C07300=1209.413,-55.510,-39.926,179.767,5.473,149.028
C07301=1209.418,-55.759,-39.914,179.765,5.472,149.029
C07302=1209.423,-56.009,-39.902,179.762,5.472,149.030
C07303=1209.429,-56.259,-39.890,179.760,5.472,149.030
C07304=1209.434,-56.509,-39.878,179.758,5.472,149.031
C07305=1209.439,-56.758,-39.867,179.755,5.471,149.032
C07306=1209.444,-57.008,-39.855,179.753,5.472,149.032
C07307=1209.449,-57.258,-39.843,179.750,5.471,149.033
C07308=1209.454,-57.508,-39.832,179.747,5.471,149.034
C07309=1209.459,-57.757,-39.819,179.745,5.471,149.035
C07310=1209.464,-58.007,-39.808,179.743,5.470,149.035
C07311=1209.470,-58.256,-39.796,179.741,5.471,149.036
C07312=1209.475,-58.506,-39.784,179.738,5.470,149.036
C07313=1209.480,-58.755,-39.773,179.736,5.470,149.037
C07314=1209.486,-59.005,-39.761,179.734,5.470,149.038
C07315=1209.491,-59.255,-39.748,179.731,5.470,149.039
C07316=1209.495,-59.504,-39.737,179.728,5.469,149.039
C07317=1209.501,-59.754,-39.725,179.726,5.470,149.040
C07318=1209.506,-60.004,-39.713,179.724,5.469,149.040
C07319=1209.511,-60.254,-39.702,179.722,5.469,149.041
C07320=1209.516,-60.504,-39.690,179.719,5.469,149.042
C07321=1209.522,-60.753,-39.679,179.717,5.468,149.043
C07322=1209.527,-61.003,-39.667,179.715,5.469,149.043
C07323=1209.533,-61.252,-39.656,179.712,5.468,149.044
C07324=1209.537,-61.501,-39.644,179.710,5.469,149.045
C07325=1209.542,-61.751,-39.632,179.707,5.468,149.045
C07326=1209.547,-62.001,-39.620,179.705,5.467,149.046
C07327=1209.552,-62.251,-39.608,179.703,5.468,149.047
C07328=1209.557,-62.501,-39.597,179.700,5.467,149.047
C07329=1209.563,-62.750,-39.586,179.698,5.468,149.048
C07330=1209.569,-63.000,-39.574,179.695,5.467,149.049
C07331=1209.573,-63.249,-39.562,179.693,5.467,149.049
C07332=1209.579,-63.499,-39.551,179.691,5.467,149.050
C07333=1209.583,-63.749,-39.539,179.688,5.467,149.051
C07334=1209.589,-63.999,-39.527,179.686,5.466,149.051
C07335=1209.594,-64.249,-39.516,179.684,5.466,149.052
C07336=1209.600,-64.498,-39.505,179.681,5.466,149.053
C07337=1209.604,-64.747,-39.493,179.679,5.466,149.053
C07338=1209.610,-64.997,-39.481,179.676,5.466,149.054
C07339=1209.614,-65.247,-39.470,179.674,5.466,149.055
C07340=1209.620,-65.497,-39.458,179.672,5.465,149.056
C07341=1209.625,-65.746,-39.447,179.669,5.465,149.056
C07342=1209.631,-65.996,-39.435,179.667,5.465,149.057
C07343=1209.635,-66.245,-39.424,179.665,5.464,149.057
C07344=1209.641,-66.495,-39.412,179.663,5.465,149.058
C07345=1209.646,-66.746,-39.402,179.660,5.464,149.059
C07346=1209.651,-66.996,-39.390,179.657,5.464,149.060
C07347=1209.656,-67.244,-39.379,179.655,5.464,149.060
C07348=1209.662,-67.494,-39.367,179.652,5.464,149.061
C07349=1209.667,-67.744,-39.356,179.650,5.464,149.062
C07350=1209.672,-67.994,-39.344,179.648,5.463,149.062
C07351=1209.677,-68.243,-39.333,179.646,5.463,149.063
C07352=1209.682,-68.492,-39.322,179.643,5.463,149.064
C07353=1209.687,-68.742,-39.310,179.641,5.463,149.064
C07354=1209.692,-68.993,-39.299,179.639,5.463,149.065
C07355=1209.698,-69.243,-39.287,179.636,5.463,149.066
C07356=1209.703,-69.492,-39.276,179.633,5.462,149.066
C07357=1209.709,-69.741,-39.264,179.632,5.462,149.067
C07358=1209.713,-69.991,-39.253,179.629,5.462,149.068
C07359=1209.718,-70.241,-39.242,179.627,5.462,149.068
C07360=1209.724,-70.491,-39.231,179.624,5.462,149.069
C07361=1209.729,-70.740,-39.220,179.622,5.462,149.070
C07362=1209.734,-70.990,-39.208,179.620,5.462,149.070
C07363=1209.739,-71.240,-39.197,179.617,5.461,149.071
C07364=1209.744,-71.489,-39.186,179.615,5.462,149.072
C07365=1209.750,-71.739,-39.175,179.613,5.461,149.072
C07366=1209.755,-71.989,-39.163,179.611,5.461,149.073
C07367=1209.761,-72.238,-39.152,179.608,5.461,149.074
C07368=1209.765,-72.488,-39.140,179.606,5.461,149.074
C07369=1209.770,-72.737,-39.129,179.603,5.461,149.075
C07370=1209.776,-72.988,-39.118,179.600,5.460,149.076
C07371=1209.781,-73.237,-39.107,179.598,5.461,149.077
C07372=1209.786,-73.486,-39.096,179.596,5.460,149.077
C07373=1209.792,-73.737,-39.085,179.594,5.460,149.078
C07374=1209.797,-73.986,-39.074,179.591,5.460,149.078
C07375=1209.802,-74.236,-39.062,179.589,5.460,149.079
C07376=1209.807,-74.485,-39.050,179.587,5.460,149.080
C07377=1209.813,-74.756,-39.039,179.584,5.459,149.081
C07378=1209.818,-75.026,-39.027,179.582,5.459,149.081
C07379=1209.824,-75.297,-39.015,179.579,5.459,149.082
C07380=1209.830,-75.568,-39.003,179.577,5.459,149.083
C07381=1209.835,-75.817,-38.992,179.575,5.459,149.083
C07382=1209.840,-76.068,-38.980,179.572,5.459,149.084
C07383=1209.846,-76.317,-38.969,179.569,5.458,149.085
C07384=1209.850,-76.566,-38.958,179.567,5.458,149.086
C07385=1209.855,-76.817,-38.948,179.565,5.458,149.086
C07386=1209.861,-77.066,-38.936,179.563,5.458,149.087
C07387=1209.866,-77.316,-38.925,179.560,5.458,149.087
C07388=1209.871,-77.566,-38.914,179.558,5.458,149.088
C07389=1209.877,-77.815,-38.903,179.555,5.457,149.089
C07390=1209.882,-78.065,-38.892,179.553,5.457,149.090
C07391=1209.887,-78.315,-38.881,179.551,5.457,149.090
C07392=1209.892,-78.564,-38.870,179.548,5.457,149.091
C07393=1209.897,-78.814,-38.859,179.546,5.457,149.091
C07394=1209.903,-79.064,-38.847,179.544,5.457,149.092
C07395=1209.908,-79.314,-38.837,179.542,5.457,149.093
C07396=1209.913,-79.563,-38.826,179.539,5.456,149.094
C07397=1209.918,-79.813,-38.816,179.537,5.457,149.094
C07398=1209.924,-80.063,-38.804,179.535,5.456,149.095
C07399=1209.929,-80.313,-38.793,179.532,5.456,149.095
C07400=1209.934,-80.562,-38.782,179.530,5.456,149.096
C07401=1209.939,-80.811,-38.771,179.527,5.455,149.097
C07402=1209.944,-81.061,-38.761,179.525,5.456,149.098
C07403=1209.950,-81.311,-38.749,179.522,5.455,149.098
C07404=1209.955,-81.561,-38.738,179.521,5.455,149.099
C07405=1209.960,-81.810,-38.727,179.518,5.455,149.099
C07406=1209.965,-82.060,-38.717,179.516,5.455,149.100
C07407=1209.970,-82.309,-38.706,179.513,5.455,149.101
C07408=1209.975,-82.559,-38.695,179.511,5.455,149.102
C07409=1209.981,-82.809,-38.683,179.509,5.455,149.102
C07410=1209.986,-83.059,-38.673,179.506,5.454,149.103
C07411=1209.991,-83.309,-38.663,179.504,5.454,149.104
C07412=1209.997,-83.558,-38.652,179.502,5.454,149.104
C07413=1210.002,-83.808,-38.641,179.500,5.454,149.105
C07414=1210.006,-84.058,-38.630,179.497,5.454,149.106
C07415=1210.012,-84.308,-38.620,179.495,5.454,149.106
C07416=1210.017,-84.557,-38.608,179.492,5.454,149.107
C07417=1210.023,-84.807,-38.598,179.491,5.454,149.108
C07418=1210.028,-85.057,-38.587,179.488,5.453,149.108
C07419=1210.033,-85.306,-38.576,179.486,5.454,149.109
C07420=1210.038,-85.556,-38.566,179.483,5.453,149.110
C07421=1210.044,-85.805,-38.555,179.481,5.453,149.110
C07422=1210.049,-86.056,-38.544,179.478,5.453,149.111
C07423=1210.054,-86.306,-38.533,179.476,5.452,149.112
C07424=1210.059,-86.555,-38.523,179.474,5.453,149.112
C07425=1210.064,-86.805,-38.512,179.471,5.452,149.113
C07426=1210.069,-87.054,-38.501,179.469,5.453,149.114
C07427=1210.074,-87.304,-38.490,179.467,5.452,149.114
C07428=1210.080,-87.554,-38.480,179.465,5.452,149.115
C07429=1210.085,-87.804,-38.468,179.462,5.452,149.116
C07430=1210.091,-88.053,-38.458,179.460,5.452,149.116
C07431=1210.096,-88.303,-38.448,179.458,5.452,149.117
C07432=1210.101,-88.552,-38.437,179.456,5.452,149.118
C07433=1210.106,-88.803,-38.426,179.453,5.452,149.118
C07434=1210.112,-89.052,-38.416,179.451,5.451,149.119
C07435=1210.117,-89.302,-38.405,179.449,5.451,149.120
C07436=1210.122,-89.551,-38.394,179.446,5.451,149.120
C07437=1210.127,-89.802,-38.384,179.444,5.451,149.121
C07438=1210.133,-90.051,-38.374,179.441,5.451,149.122
C07439=1210.137,-90.301,-38.362,179.439,5.451,149.122
C07440=1210.143,-90.550,-38.352,179.437,5.450,149.123
C07441=1210.148,-90.801,-38.341,179.435,5.451,149.124
C07442=1210.154,-91.050,-38.331,179.432,5.450,149.124
C07443=1210.158,-91.300,-38.320,179.430,5.451,149.125
C07444=1210.164,-91.549,-38.310,179.427,5.450,149.126
C07445=1210.169,-91.800,-38.299,179.426,5.450,149.126
C07446=1210.174,-92.049,-38.289,179.423,5.450,149.127
C07447=1210.179,-92.299,-38.278,179.421,5.450,149.128
C07448=1210.185,-92.548,-38.268,179.418,5.450,149.128
C07449=1210.190,-92.798,-38.257,179.416,5.450,149.129
C07450=1210.195,-93.048,-38.247,179.414,5.449,149.130
C07451=1210.200,-93.297,-38.237,179.412,5.450,149.130
C07452=1210.205,-93.547,-38.227,179.409,5.449,149.131
C07453=1210.210,-93.796,-38.216,179.407,5.449,149.132
C07454=1210.215,-94.047,-38.205,179.405,5.449,149.132
C07455=1210.221,-94.296,-38.195,179.402,5.449,149.133
C07456=1210.226,-94.546,-38.184,179.400,5.449,149.134
C07457=1210.232,-94.796,-38.174,179.398,5.448,149.134
C07458=1210.237,-95.046,-38.164,179.396,5.449,149.135
C07459=1210.242,-95.296,-38.153,179.393,5.448,149.136
C07460=1210.248,-95.545,-38.142,179.391,5.449,149.137
C07461=1210.253,-95.795,-38.132,179.389,5.448,149.137
C07462=1210.258,-96.044,-38.122,179.387,5.448,149.138
C07463=1210.263,-96.294,-38.112,179.384,5.448,149.138
C07464=1210.268,-96.544,-38.101,179.382,5.448,149.139
C07465=1210.274,-96.793,-38.091,179.379,5.448,149.140
C07466=1210.279,-97.044,-38.081,179.377,5.448,149.140
C07467=1210.284,-97.293,-38.070,179.375,5.447,149.141
C07468=1210.290,-97.543,-38.060,179.373,5.448,149.142
C07469=1210.295,-97.793,-38.050,179.370,5.447,149.142
C07470=1210.300,-98.043,-38.039,179.368,5.448,149.143
C07471=1210.305,-98.293,-38.029,179.366,5.447,149.144
C07472=1210.310,-98.541,-38.018,179.364,5.447,149.144
C07473=1210.316,-98.791,-38.008,179.361,5.447,149.145
C07474=1210.321,-99.041,-37.998,179.359,5.447,149.146
C07475=1210.326,-99.291,-37.987,179.357,5.446,149.146
C07476=1210.332,-99.540,-37.977,179.355,5.447,149.147
C07477=1210.336,-99.790,-37.967,179.352,5.446,149.148
C07478=1210.342,-100.040,-37.957,179.350,5.447,149.148
C07479=1210.347,-100.289,-37.947,179.347,5.446,149.149
C07480=1210.352,-100.540,-37.936,179.346,5.446,149.150
C07481=1210.357,-100.811,-37.925,179.343,5.446,149.150
C07482=1210.364,-101.082,-37.914,179.340,5.445,149.151
C07483=1210.369,-101.353,-37.903,179.338,5.446,149.152
C07484=1210.375,-101.625,-37.892,179.335,5.446,149.153
C07485=1210.380,-101.875,-37.883,179.333,5.446,149.153
C07486=1210.386,-102.124,-37.873,179.331,5.445,149.154
C07487=1210.391,-102.374,-37.862,179.329,5.446,149.155
C07488=1210.396,-102.624,-37.852,179.326,5.445,149.155
C07489=1210.401,-102.873,-37.842,179.324,5.445,149.156
C07490=1210.406,-103.123,-37.832,179.322,5.445,149.157
C07491=1210.412,-103.373,-37.821,179.320,5.445,149.157
C07492=1210.417,-103.622,-37.811,179.317,5.445,149.158
C07493=1210.422,-103.872,-37.801,179.315,5.445,149.159
C07494=1210.427,-104.122,-37.791,179.313,5.444,149.159
C07495=1210.433,-104.371,-37.781,179.311,5.445,149.160
C07496=1210.438,-104.622,-37.771,179.308,5.444,149.161
C07497=1210.443,-104.872,-37.761,179.306,5.445,149.161
C07498=1210.449,-105.121,-37.751,179.304,5.444,149.162
C07499=1210.454,-105.371,-37.741,179.302,5.444,149.162
C07500=1210.458,-105.621,-37.731,179.299,5.444,149.163
C07501=1210.464,-105.870,-37.721,179.297,5.444,149.164
C07502=1210.470,-106.120,-37.711,179.295,5.444,149.164
C07503=1210.475,-106.371,-37.701,179.292,5.444,149.165
C07504=1210.480,-106.620,-37.691,179.290,5.444,149.166
C07505=1210.485,-106.869,-37.681,179.288,5.444,149.167
C07506=1210.491,-107.119,-37.671,179.285,5.444,149.167
C07507=1210.495,-107.369,-37.661,179.283,5.444,149.168
C07508=1210.501,-107.618,-37.650,179.281,5.443,149.168
C07509=1210.507,-107.869,-37.641,179.279,5.443,149.169
C07510=1210.512,-108.118,-37.631,179.276,5.443,149.170
C07511=1210.517,-108.368,-37.621,179.274,5.443,149.170
C07512=1210.522,-108.618,-37.611,179.272,5.443,149.171
C07513=1210.527,-108.867,-37.602,179.270,5.443,149.172
C07514=1210.533,-109.117,-37.591,179.267,5.443,149.173
C07515=1210.537,-109.367,-37.581,179.265,5.443,149.173
C07516=1210.543,-109.616,-37.571,179.263,5.442,149.174
C07517=1210.549,-109.867,-37.562,179.261,5.443,149.174
C07518=1210.554,-110.116,-37.552,179.258,5.442,149.175
C07519=1210.559,-110.365,-37.542,179.256,5.442,149.176
C07520=1210.564,-110.616,-37.531,179.254,5.442,149.176
C07521=1210.569,-110.865,-37.522,179.252,5.442,149.177
C07522=1210.575,-111.115,-37.512,179.249,5.442,149.178
C07523=1210.580,-111.364,-37.503,179.247,5.442,149.178
C07524=1210.585,-111.615,-37.493,179.245,5.441,149.179
C07525=1210.591,-111.865,-37.483,179.242,5.442,149.180
C07526=1210.596,-112.114,-37.473,179.240,5.441,149.180
C07527=1210.602,-112.364,-37.463,179.238,5.441,149.181
C07528=1210.606,-112.613,-37.454,179.236,5.441,149.182
C07529=1210.612,-112.863,-37.444,179.233,5.441,149.182
C07530=1210.617,-113.113,-37.434,179.231,5.441,149.183
C07531=1210.622,-113.363,-37.424,179.229,5.441,149.184
C07532=1210.628,-113.612,-37.414,179.227,5.441,149.184
C07533=1210.633,-113.862,-37.405,179.224,5.441,149.185
C07534=1210.639,-114.112,-37.395,179.222,5.441,149.186
C07535=1210.643,-114.362,-37.385,179.220,5.440,149.186
C07536=1210.649,-114.612,-37.375,179.218,5.441,149.187
C07537=1210.654,-114.861,-37.366,179.215,5.440,149.188
C07538=1210.659,-115.111,-37.356,179.213,5.441,149.188
C07539=1210.664,-115.361,-37.347,179.211,5.440,149.189
C07540=1210.670,-115.610,-37.336,179.209,5.440,149.189
C07541=1210.675,-115.860,-37.328,179.206,5.440,149.190
C07542=1210.680,-116.110,-37.317,179.205,5.440,149.191
C07543=1210.685,-116.360,-37.308,179.202,5.440,149.191
C07544=1210.691,-116.610,-37.298,179.200,5.440,149.192
C07545=1210.696,-116.859,-37.289,179.197,5.440,149.193
C07546=1210.702,-117.109,-37.279,179.196,5.440,149.193
C07547=1210.707,-117.359,-37.270,179.193,5.439,149.194
C07548=1210.712,-117.608,-37.260,179.191,5.440,149.195
C07549=1210.717,-117.858,-37.250,179.188,5.439,149.195
C07550=1210.723,-118.108,-37.240,179.187,5.439,149.196
C07551=1210.727,-118.358,-37.231,179.184,5.440,149.197
C07552=1210.733,-118.608,-37.221,179.182,5.439,149.197
C07553=1210.738,-118.857,-37.212,179.180,5.439,149.198
C07554=1210.743,-119.107,-37.203,179.178,5.439,149.199
C07555=1210.749,-119.356,-37.192,179.175,5.439,149.199
C07556=1210.754,-119.606,-37.183,179.173,5.439,149.200
C07557=1210.760,-119.856,-37.173,179.171,5.439,149.201
C07558=1210.764,-120.106,-37.164,179.168,5.438,149.201
C07559=1210.770,-120.357,-37.155,179.166,5.439,149.202
C07560=1210.775,-120.606,-37.145,179.164,5.438,149.202
C07561=1210.780,-120.856,-37.136,179.162,5.438,149.203
C07562=1210.786,-121.105,-37.126,179.159,5.438,149.204
C07563=1210.791,-121.355,-37.117,179.157,5.438,149.205
C07564=1210.797,-121.605,-37.107,179.155,5.437,149.205
C07565=1210.802,-121.854,-37.098,179.153,5.438,149.206
C07566=1210.807,-122.104,-37.088,179.151,5.438,149.207
C07567=1210.812,-122.354,-37.079,179.149,5.437,149.207
C07568=1210.818,-122.604,-37.070,179.147,5.438,149.208
C07569=1210.823,-122.853,-37.060,179.144,5.437,149.208
C07570=1210.828,-123.103,-37.051,179.142,5.437,149.209
C07571=1210.833,-123.354,-37.041,179.140,5.437,149.210
C07572=1210.839,-123.603,-37.031,179.138,5.437,149.210
C07573=1210.844,-123.853,-37.022,179.135,5.437,149.211
C07574=1210.849,-124.102,-37.013,179.133,5.437,149.212
C07575=1210.854,-124.352,-37.003,179.131,5.437,149.212
C07576=1210.860,-124.602,-36.994,179.129,5.437,149.213
C07577=1210.865,-124.852,-36.985,179.126,5.436,149.213
C07578=1210.870,-125.102,-36.975,179.124,5.437,149.214
C07579=1210.876,-125.352,-36.966,179.122,5.437,149.215
C07580=1210.880,-125.601,-36.957,179.120,5.436,149.215
C07581=1210.886,-125.851,-36.947,179.118,5.437,149.216
C07582=1210.892,-126.101,-36.938,179.115,5.436,149.217
C07583=1210.896,-126.350,-36.929,179.113,5.437,149.218
C07584=1210.902,-126.600,-36.919,179.111,5.436,149.218
C07585=1210.481,-126.611,-36.957,179.107,5.439,149.220
C07586=1210.476,-126.361,-36.966,179.109,5.440,149.219
C07587=1210.471,-126.111,-36.976,179.111,5.439,149.219
C07588=1210.465,-125.861,-36.985,179.113,5.440,149.218
C07589=1210.460,-125.611,-36.994,179.116,5.440,149.217
C07590=1210.455,-125.362,-37.004,179.118,5.440,149.217
C07591=1210.449,-125.112,-37.013,179.120,5.440,149.216
C07592=1210.444,-124.862,-37.022,179.122,5.440,149.216
C07593=1210.439,-124.613,-37.032,179.125,5.440,149.215
C07594=1210.433,-124.363,-37.041,179.127,5.440,149.214
C07595=1210.428,-124.113,-37.050,179.129,5.441,149.214
C07596=1210.423,-123.864,-37.060,179.131,5.440,149.213
C07597=1210.417,-123.614,-37.069,179.134,5.441,149.212
C07598=1210.412,-123.364,-37.078,179.135,5.441,149.212
C07599=1210.407,-123.114,-37.088,179.138,5.441,149.211
C07600=1210.401,-122.864,-37.097,179.140,5.441,149.210
C07601=1210.396,-122.614,-37.106,179.142,5.441,149.210
C07602=1210.390,-122.365,-37.116,179.144,5.441,149.209
C07603=1210.385,-122.115,-37.125,179.147,5.441,149.208
C07604=1210.380,-121.866,-37.135,179.149,5.441,149.208
C07605=1210.374,-121.616,-37.144,179.151,5.441,149.207
C07606=1210.369,-121.366,-37.154,179.153,5.441,149.206
C07607=1210.365,-121.116,-37.163,179.155,5.441,149.206
C07608=1210.359,-120.866,-37.173,179.158,5.442,149.205
C07609=1210.354,-120.616,-37.182,179.160,5.441,149.205
C07610=1210.348,-120.366,-37.192,179.162,5.442,149.204
C07611=1210.343,-120.117,-37.201,179.165,5.441,149.203
C07612=1210.337,-119.867,-37.211,179.167,5.442,149.203
C07613=1210.333,-119.618,-37.221,179.169,5.442,149.202
C07614=1210.327,-119.368,-37.229,179.172,5.442,149.201
C07615=1210.322,-119.118,-37.240,179.173,5.442,149.201
C07616=1210.317,-118.868,-37.249,179.176,5.443,149.200
C07617=1210.311,-118.619,-37.259,179.178,5.442,149.199
C07618=1210.307,-118.368,-37.268,179.181,5.443,149.199
C07619=1210.301,-118.119,-37.278,179.182,5.443,149.198
C07620=1210.296,-117.869,-37.287,179.184,5.442,149.197
C07621=1210.290,-117.619,-37.297,179.187,5.443,149.197
C07622=1210.285,-117.370,-37.306,179.189,5.443,149.196
C07623=1210.280,-117.120,-37.316,179.191,5.443,149.195
C07624=1210.274,-116.870,-37.325,179.193,5.443,149.195
C07625=1210.269,-116.621,-37.335,179.196,5.443,149.194
C07626=1210.264,-116.370,-37.345,179.198,5.443,149.194
C07627=1210.259,-116.121,-37.354,179.200,5.444,149.193
C07628=1210.254,-115.871,-37.365,179.202,5.443,149.192
C07629=1210.248,-115.621,-37.374,179.205,5.444,149.192
C07630=1210.243,-115.372,-37.384,179.207,5.444,149.191
C07631=1210.238,-115.122,-37.393,179.209,5.444,149.190
C07632=1210.233,-114.872,-37.403,179.211,5.444,149.189
C07633=1210.227,-114.622,-37.413,179.214,5.444,149.189
C07634=1210.222,-114.372,-37.422,179.216,5.444,149.188
C07635=1210.216,-114.123,-37.433,179.218,5.444,149.188
C07636=1210.211,-113.873,-37.441,179.220,5.444,149.187
C07637=1210.206,-113.623,-37.452,179.223,5.445,149.186
C07638=1210.201,-113.374,-37.461,179.225,5.444,149.186
C07639=1210.195,-113.123,-37.471,179.227,5.445,149.185
C07640=1210.191,-112.874,-37.481,179.229,5.444,149.184
C07641=1210.185,-112.624,-37.490,179.231,5.444,149.184
C07642=1210.179,-112.374,-37.500,179.234,5.445,149.183
C07643=1210.174,-112.125,-37.510,179.236,5.444,149.182
C07644=1210.169,-111.874,-37.520,179.239,5.445,149.182
C07645=1210.164,-111.625,-37.530,179.240,5.445,149.181
C07646=1210.158,-111.376,-37.540,179.243,5.445,149.180
C07647=1210.154,-111.126,-37.549,179.245,5.445,149.180
C07648=1210.148,-110.876,-37.559,179.247,5.446,149.179
C07649=1210.143,-110.626,-37.569,179.249,5.445,149.178
C07650=1210.138,-110.377,-37.579,179.252,5.446,149.178
C07651=1210.132,-110.127,-37.589,179.254,5.445,149.177
C07652=1210.127,-109.877,-37.598,179.256,5.446,149.177
C07653=1210.122,-109.627,-37.609,179.258,5.446,149.176
C07654=1210.116,-109.378,-37.619,179.261,5.446,149.175
C07655=1210.111,-109.128,-37.628,179.263,5.446,149.174
C07656=1210.106,-108.878,-37.638,179.265,5.447,149.174
C07657=1210.100,-108.629,-37.648,179.267,5.446,149.173
C07658=1210.096,-108.379,-37.658,179.270,5.447,149.172
C07659=1210.090,-108.128,-37.668,179.272,5.446,149.172
C07660=1210.084,-107.879,-37.678,179.275,5.447,149.171
C07661=1210.079,-107.630,-37.688,179.276,5.447,149.171
C07662=1210.074,-107.379,-37.698,179.279,5.447,149.170
C07663=1210.069,-107.130,-37.708,179.281,5.447,149.169
C07664=1210.064,-106.880,-37.717,179.284,5.447,149.168
C07665=1210.058,-106.631,-37.727,179.285,5.447,149.168
C07666=1210.053,-106.380,-37.738,179.288,5.448,149.167
C07667=1210.048,-106.131,-37.748,179.290,5.447,149.167
C07668=1210.043,-105.882,-37.758,179.293,5.448,149.166
C07669=1210.037,-105.631,-37.768,179.294,5.448,149.165
C07670=1210.032,-105.381,-37.777,179.297,5.448,149.165
C07671=1210.027,-105.132,-37.788,179.299,5.448,149.164
C07672=1210.021,-104.882,-37.798,179.302,5.448,149.163
C07673=1210.017,-104.632,-37.808,179.303,5.448,149.163
C07674=1210.011,-104.383,-37.818,179.306,5.448,149.162
C07675=1210.006,-104.133,-37.828,179.308,5.448,149.161
C07676=1210.001,-103.883,-37.839,179.311,5.448,149.161
C07677=1209.996,-103.633,-37.848,179.313,5.448,149.160
C07678=1209.990,-103.384,-37.858,179.315,5.449,149.159
C07679=1209.985,-103.133,-37.868,179.317,5.448,149.159
C07680=1209.979,-102.884,-37.879,179.320,5.449,149.158
C07681=1209.975,-102.635,-37.888,179.322,5.449,149.157
C07682=1209.970,-102.384,-37.899,179.324,5.449,149.157
C07683=1209.964,-102.135,-37.909,179.326,5.449,149.156
C07684=1209.958,-101.885,-37.919,179.329,5.449,149.155
C07685=1209.954,-101.635,-37.929,179.331,5.449,149.155
C07686=1209.948,-101.364,-37.940,179.334,5.449,149.154
C07687=1209.942,-101.093,-37.951,179.336,5.449,149.153
C07688=1209.936,-100.822,-37.963,179.338,5.449,149.152
C07689=1209.931,-100.551,-37.973,179.341,5.450,149.152
C07690=1209.926,-100.301,-37.984,179.343,5.449,149.151
C07691=1209.920,-100.051,-37.994,179.345,5.450,149.151
C07692=1209.915,-99.802,-38.004,179.348,5.450,149.150
C07693=1209.910,-99.552,-38.014,179.350,5.450,149.149
C07694=1209.905,-99.302,-38.025,179.352,5.450,149.148
C07695=1209.900,-99.052,-38.035,179.355,5.450,149.148
C07696=1209.894,-98.802,-38.045,179.357,5.450,149.147
C07697=1209.888,-98.553,-38.056,179.359,5.451,149.146
C07698=1209.884,-98.303,-38.066,179.361,5.450,149.146
C07699=1209.879,-98.053,-38.076,179.364,5.451,149.145
C07700=1209.873,-97.804,-38.086,179.366,5.451,149.145
C07701=1209.868,-97.554,-38.097,179.368,5.451,149.144
C07702=1209.862,-97.304,-38.107,179.370,5.451,149.143
C07703=1209.857,-97.054,-38.117,179.373,5.451,149.142
C07704=1209.852,-96.804,-38.128,179.375,5.451,149.142
C07705=1209.846,-96.555,-38.138,179.377,5.452,149.141
C07706=1209.842,-96.305,-38.148,179.379,5.451,149.141
C07707=1209.836,-96.055,-38.158,179.382,5.452,149.140
C07708=1209.831,-95.805,-38.168,179.384,5.451,149.139
C07709=1209.826,-95.556,-38.179,179.387,5.452,149.138
C07710=1209.820,-95.307,-38.190,179.388,5.452,149.138
C07711=1209.815,-95.056,-38.200,179.391,5.452,149.137
C07712=1209.810,-94.807,-38.210,179.393,5.452,149.136
C07713=1209.805,-94.556,-38.221,179.396,5.452,149.136
C07714=1209.799,-94.307,-38.231,179.399,5.453,149.135
C07715=1209.794,-94.057,-38.241,179.400,5.453,149.135
C07716=1209.789,-93.807,-38.252,179.403,5.453,149.134
C07717=1209.784,-93.559,-38.262,179.405,5.453,149.133
C07718=1209.779,-93.308,-38.273,179.408,5.453,149.132
C07719=1209.774,-93.059,-38.283,179.410,5.453,149.132
C07720=1209.769,-92.808,-38.294,179.412,5.454,149.131
C07721=1209.763,-92.559,-38.304,179.414,5.453,149.131
C07722=1209.758,-92.309,-38.315,179.417,5.454,149.130
C07723=1209.753,-92.060,-38.325,179.419,5.453,149.129
C07724=1209.747,-91.810,-38.336,179.421,5.454,149.128
C07725=1209.742,-91.560,-38.346,179.423,5.453,149.128
C07726=1209.736,-91.310,-38.356,179.426,5.454,149.127
C07727=1209.732,-91.061,-38.368,179.428,5.454,149.127
C07728=1209.726,-90.811,-38.378,179.430,5.454,149.126
C07729=1209.721,-90.561,-38.388,179.433,5.454,149.125
C07730=1209.716,-90.312,-38.399,179.435,5.454,149.124
C07731=1209.711,-90.062,-38.410,179.437,5.454,149.124
C07732=1209.705,-89.812,-38.420,179.439,5.455,149.123
C07733=1209.700,-89.562,-38.431,179.442,5.454,149.122
C07734=1209.695,-89.313,-38.441,179.444,5.455,149.122
C07735=1209.690,-89.063,-38.452,179.447,5.455,149.121
C07736=1209.684,-88.813,-38.462,179.448,5.455,149.121
C07737=1209.679,-88.563,-38.473,179.451,5.456,149.120
C07738=1209.674,-88.314,-38.484,179.453,5.455,149.119
C07739=1209.669,-88.064,-38.494,179.456,5.456,149.118
C07740=1209.663,-87.814,-38.505,179.458,5.455,149.118
C07741=1209.659,-87.565,-38.516,179.461,5.456,149.117
C07742=1209.653,-87.315,-38.526,179.462,5.456,149.117
C07743=1209.648,-87.065,-38.537,179.465,5.456,149.116
C07744=1209.643,-86.816,-38.548,179.467,5.456,149.115
C07745=1209.637,-86.566,-38.559,179.470,5.456,149.114
C07746=1209.632,-86.316,-38.569,179.472,5.456,149.114
C07747=1209.627,-86.066,-38.580,179.474,5.456,149.113
C07748=1209.622,-85.816,-38.591,179.477,5.457,149.112
C07749=1209.617,-85.567,-38.602,179.479,5.457,149.112
C07750=1209.612,-85.317,-38.612,179.481,5.457,149.111
C07751=1209.606,-85.067,-38.623,179.484,5.457,149.110
C07752=1209.601,-84.818,-38.634,179.486,5.457,149.110
C07753=1209.596,-84.568,-38.644,179.488,5.457,149.109
C07754=1209.591,-84.319,-38.655,179.490,5.458,149.108
C07755=1209.585,-84.069,-38.666,179.493,5.457,149.108
C07756=1209.580,-83.818,-38.677,179.495,5.458,149.107
C07757=1209.575,-83.569,-38.688,179.497,5.457,149.106
C07758=1209.569,-83.319,-38.698,179.500,5.458,149.106
C07759=1209.565,-83.070,-38.710,179.502,5.459,149.105
C07760=1209.559,-82.820,-38.720,179.504,5.458,149.104
C07761=1209.554,-82.571,-38.731,179.507,5.459,149.104
C07762=1209.549,-82.321,-38.741,179.509,5.458,149.103
C07763=1209.543,-82.071,-38.753,179.512,5.459,149.102
C07764=1209.538,-81.821,-38.764,179.514,5.458,149.102
C07765=1209.533,-81.572,-38.775,179.516,5.459,149.101
C07766=1209.528,-81.322,-38.785,179.518,5.459,149.100
C07767=1209.523,-81.073,-38.796,179.521,5.459,149.100
C07768=1209.518,-80.822,-38.807,179.523,5.460,149.099
C07769=1209.512,-80.573,-38.819,179.525,5.459,149.098
C07770=1209.507,-80.323,-38.829,179.528,5.460,149.098
C07771=1209.502,-80.073,-38.840,179.530,5.459,149.097
C07772=1209.497,-79.823,-38.851,179.532,5.460,149.096
C07773=1209.492,-79.574,-38.862,179.534,5.460,149.096
C07774=1209.486,-79.324,-38.873,179.537,5.460,149.095
C07775=1209.481,-79.075,-38.884,179.539,5.460,149.094
C07776=1209.476,-78.825,-38.895,179.542,5.460,149.094
C07777=1209.471,-78.575,-38.906,179.545,5.461,149.093
C07778=1209.465,-78.326,-38.917,179.546,5.461,149.092
C07779=1209.460,-78.075,-38.928,179.549,5.461,149.092
C07780=1209.455,-77.826,-38.939,179.551,5.461,149.091
C07781=1209.450,-77.577,-38.950,179.554,5.461,149.090
C07782=1209.444,-77.326,-38.961,179.556,5.461,149.090
C07783=1209.440,-77.077,-38.972,179.558,5.461,149.089
C07784=1209.434,-76.827,-38.983,179.560,5.462,149.088
C07785=1209.429,-76.577,-38.994,179.563,5.462,149.088
C07786=1209.424,-76.328,-39.006,179.565,5.462,149.087
C07787=1209.418,-76.078,-39.016,179.567,5.462,149.086
C07788=1209.414,-75.828,-39.027,179.570,5.462,149.085
C07789=1209.408,-75.579,-39.039,179.572,5.462,149.085
C07790=1209.403,-75.308,-39.050,179.575,5.463,149.084
C07791=1209.397,-75.037,-39.063,179.578,5.463,149.083
C07792=1209.391,-74.767,-39.075,179.580,5.463,149.083
C07793=1209.385,-74.496,-39.087,179.582,5.463,149.082
C07794=1209.381,-74.247,-39.098,179.585,5.463,149.081
C07795=1209.375,-73.997,-39.108,179.587,5.463,149.081
C07796=1209.370,-73.747,-39.120,179.590,5.464,149.080
C07797=1209.365,-73.498,-39.131,179.592,5.463,149.079
C07798=1209.360,-73.248,-39.143,179.594,5.464,149.079
C07799=1209.354,-72.998,-39.154,179.597,5.464,149.078
C07800=1209.349,-72.748,-39.165,179.599,5.464,149.077
C07801=1209.344,-72.498,-39.177,179.601,5.465,149.077
C07802=1209.338,-72.249,-39.187,179.603,5.464,149.076
C07803=1209.333,-71.999,-39.198,179.606,5.465,149.075
C07804=1209.328,-71.749,-39.210,179.608,5.465,149.075
C07805=1209.323,-71.500,-39.221,179.610,5.465,149.074
C07806=1209.318,-71.251,-39.232,179.613,5.466,149.073
C07807=1209.312,-71.000,-39.244,179.615,5.465,149.072
C07808=1209.308,-70.751,-39.255,179.618,5.466,149.072
C07809=1209.302,-70.501,-39.266,179.620,5.465,149.071
C07810=1209.297,-70.252,-39.278,179.623,5.466,149.070
C07811=1209.292,-70.002,-39.289,179.625,5.465,149.070
C07812=1209.286,-69.752,-39.300,179.627,5.466,149.069
C07813=1209.281,-69.503,-39.311,179.630,5.467,149.068
C07814=1209.276,-69.253,-39.323,179.632,5.466,149.068
C07815=1209.271,-69.003,-39.334,179.634,5.467,149.067
C07816=1209.266,-68.753,-39.346,179.636,5.466,149.066
C07817=1209.261,-68.504,-39.357,179.639,5.467,149.066
C07818=1209.255,-68.254,-39.368,179.642,5.467,149.065
C07819=1209.250,-68.004,-39.379,179.643,5.467,149.064
C07820=1209.245,-67.754,-39.391,179.646,5.468,149.064
C07821=1209.240,-67.504,-39.403,179.648,5.467,149.063
C07822=1209.234,-67.256,-39.414,179.651,5.468,149.062
C07823=1209.229,-67.006,-39.425,179.653,5.468,149.062
C07824=1209.224,-66.756,-39.437,179.655,5.468,149.061
C07825=1209.219,-66.506,-39.449,179.658,5.468,149.060
C07826=1209.214,-66.256,-39.460,179.660,5.468,149.060
C07827=1209.208,-66.007,-39.471,179.662,5.469,149.059
C07828=1209.203,-65.758,-39.483,179.665,5.469,149.058
C07829=1209.198,-65.508,-39.495,179.667,5.469,149.058
C07830=1209.193,-65.257,-39.505,179.670,5.469,149.057
C07831=1209.188,-65.007,-39.517,179.672,5.469,149.056
C07832=1209.183,-64.758,-39.528,179.675,5.469,149.056
C07833=1209.177,-64.509,-39.540,179.677,5.470,149.055
C07834=1209.172,-64.259,-39.551,179.679,5.470,149.054
C07835=1209.167,-64.009,-39.563,179.682,5.470,149.054
C07836=1209.162,-63.759,-39.574,179.684,5.470,149.053
C07837=1209.157,-63.509,-39.586,179.686,5.470,149.052
C07838=1209.152,-63.260,-39.598,179.689,5.471,149.052
C07839=1209.146,-63.011,-39.609,179.691,5.471,149.051
C07840=1209.141,-62.761,-39.620,179.694,5.471,149.050
C07841=1209.136,-62.511,-39.632,179.696,5.471,149.049
C07842=1209.131,-62.261,-39.644,179.698,5.471,149.049
C07843=1209.126,-62.012,-39.656,179.701,5.472,149.048
C07844=1209.121,-61.762,-39.668,179.703,5.472,149.048
C07845=1209.116,-61.513,-39.679,179.705,5.472,149.047
C07846=1209.110,-61.263,-39.691,179.707,5.472,149.046
C07847=1209.105,-61.014,-39.702,179.710,5.472,149.045
C07848=1209.100,-60.764,-39.714,179.713,5.473,149.045
C07849=1209.094,-60.514,-39.726,179.715,5.472,149.044
C07850=1209.090,-60.264,-39.737,179.717,5.473,149.043
C07851=1209.084,-60.014,-39.749,179.719,5.473,149.043
C07852=1209.080,-59.765,-39.760,179.722,5.473,149.042
C07853=1209.074,-59.515,-39.772,179.724,5.474,149.041
C07854=1209.069,-59.265,-39.785,179.727,5.473,149.041
C07855=1209.064,-59.016,-39.796,179.729,5.474,149.040
C07856=1209.058,-58.767,-39.808,179.732,5.474,149.039
C07857=1209.054,-58.517,-39.819,179.734,5.474,149.039
C07858=1209.048,-58.267,-39.831,179.736,5.475,149.038
C07859=1209.043,-58.017,-39.843,179.738,5.474,149.037
C07860=1209.038,-57.767,-39.854,179.741,5.475,149.037
C07861=1209.033,-57.518,-39.867,179.744,5.475,149.036
C07862=1209.027,-57.268,-39.878,179.746,5.475,149.035
C07863=1209.023,-57.019,-39.890,179.748,5.475,149.035
C07864=1209.017,-56.769,-39.902,179.750,5.475,149.034
C07865=1209.012,-56.519,-39.914,179.753,5.475,149.033
C07866=1209.007,-56.270,-39.926,179.755,5.476,149.033
C07867=1209.002,-56.020,-39.937,179.757,5.476,149.032
C07868=1208.997,-55.770,-39.949,179.760,5.476,149.031
C07869=1208.992,-55.520,-39.961,179.763,5.477,149.031
C07870=1208.987,-55.271,-39.973,179.765,5.476,149.030
C07871=1208.981,-55.022,-39.985,179.767,5.477,149.029
C07872=1208.975,-54.772,-39.997,179.770,5.477,149.028
C07873=1208.971,-54.522,-40.008,179.772,5.477,149.028
C07874=1208.966,-54.273,-40.020,179.775,5.477,149.027
C07875=1208.960,-54.023,-40.032,179.776,5.477,149.027
C07876=1208.955,-53.773,-40.044,179.779,5.478,149.026
C07877=1208.950,-53.523,-40.056,179.782,5.478,149.025
C07878=1208.945,-53.274,-40.068,179.784,5.478,149.024
C07879=1208.939,-53.024,-40.080,179.787,5.479,149.024
C07880=1208.935,-52.774,-40.091,179.789,5.479,149.023
C07881=1208.930,-52.525,-40.104,179.791,5.479,149.022
C07882=1208.924,-52.275,-40.116,179.794,5.479,149.022
C07883=1208.919,-52.025,-40.128,179.796,5.479,149.021
C07884=1208.914,-51.776,-40.140,179.798,5.480,149.020
C07885=1208.909,-51.526,-40.152,179.801,5.480,149.020
C07886=1208.904,-51.276,-40.163,179.803,5.480,149.019
C07887=1208.898,-51.027,-40.176,179.806,5.480,149.018
C07888=1208.893,-50.777,-40.188,179.808,5.481,149.018
C07889=1208.889,-50.528,-40.200,179.810,5.480,149.017
C07890=1208.883,-50.278,-40.212,179.813,5.481,149.016
C07891=1208.878,-50.028,-40.224,179.816,5.481,149.016
C07892=1208.873,-49.779,-40.236,179.817,5.481,149.015
C07893=1208.868,-49.528,-40.249,179.820,5.482,149.014
C07894=1208.862,-49.259,-40.261,179.823,5.482,149.014
C07895=1208.857,-48.989,-40.275,179.825,5.481,149.013
C07896=1208.851,-48.719,-40.287,179.828,5.482,149.012
C07897=1208.846,-48.449,-40.300,179.831,5.482,149.011
C07898=1208.841,-48.199,-40.313,179.833,5.483,149.011
C07899=1208.835,-47.950,-40.325,179.835,5.482,149.010
C07900=1208.830,-47.700,-40.337,179.838,5.483,149.009
C07901=1208.825,-47.450,-40.349,179.840,5.484,149.009
C07902=1208.819,-47.200,-40.361,179.842,5.483,149.008
C07903=1208.814,-46.951,-40.374,179.845,5.484,149.007
C07904=1208.809,-46.701,-40.386,179.848,5.484,149.007
C07905=1208.805,-46.451,-40.398,179.850,5.484,149.006
C07906=1208.799,-46.201,-40.410,179.852,5.484,149.005
C07907=1208.794,-45.952,-40.423,179.855,5.485,149.005
C07908=1208.789,-45.702,-40.435,179.857,5.485,149.004
C07909=1208.784,-45.453,-40.447,179.860,5.485,149.003
C07910=1208.778,-45.203,-40.459,179.862,5.486,149.003
C07911=1208.773,-44.954,-40.472,179.864,5.486,149.002
C07912=1208.768,-44.704,-40.484,179.867,5.486,149.001
C07913=1208.763,-44.454,-40.496,179.869,5.486,149.001
C07914=1208.757,-44.205,-40.509,179.871,5.486,149.000
C07915=1208.753,-43.954,-40.521,179.874,5.487,148.999
C07916=1208.747,-43.705,-40.534,179.877,5.487,148.998
C07917=1208.742,-43.455,-40.545,179.879,5.487,148.998
C07918=1208.738,-43.206,-40.557,179.881,5.487,148.997
C07919=1208.733,-42.957,-40.570,179.884,5.488,148.997
C07920=1208.727,-42.707,-40.582,179.886,5.488,148.996
C07921=1208.722,-42.458,-40.595,179.888,5.488,148.995
C07922=1208.717,-42.208,-40.606,179.891,5.489,148.994
C07923=1208.712,-41.958,-40.619,179.893,5.488,148.994
C07924=1208.707,-41.708,-40.632,179.896,5.489,148.993
C07925=1208.701,-41.458,-40.644,179.898,5.489,148.992
C07926=1208.696,-41.209,-40.656,179.901,5.489,148.992
C07927=1208.691,-40.960,-40.669,179.903,5.489,148.991
C07928=1208.686,-40.710,-40.681,179.906,5.490,148.990
C07929=1208.681,-40.460,-40.694,179.907,5.490,148.990
C07930=1208.676,-40.210,-40.707,179.910,5.490,148.989
C07931=1208.671,-39.961,-40.718,179.913,5.491,148.988
C07932=1208.666,-39.711,-40.731,179.915,5.490,148.988
C07933=1208.660,-39.462,-40.744,179.918,5.491,148.987
C07934=1208.654,-39.212,-40.756,179.920,5.491,148.986
C07935=1208.650,-38.962,-40.769,179.922,5.491,148.986
C07936=1208.645,-38.712,-40.782,179.925,5.491,148.985
C07937=1208.640,-38.463,-40.794,179.928,5.492,148.984
C07938=1208.634,-38.213,-40.806,179.929,5.492,148.984
C07939=1208.629,-37.964,-40.819,179.932,5.492,148.983
C07940=1208.624,-37.714,-40.831,179.934,5.493,148.982
C07941=1208.619,-37.464,-40.844,179.937,5.493,148.982
C07942=1208.614,-37.214,-40.856,179.939,5.493,148.981
C07943=1208.609,-36.965,-40.869,179.942,5.494,148.980
C07944=1208.604,-36.716,-40.881,179.945,5.494,148.980
C07945=1208.599,-36.466,-40.894,179.947,5.494,148.979
C07946=1208.593,-36.216,-40.908,179.949,5.494,148.978
C07947=1208.588,-35.966,-40.919,179.952,5.495,148.977
C07948=1208.583,-35.717,-40.932,179.954,5.495,148.977
C07949=1208.578,-35.468,-40.945,179.956,5.495,148.976
C07950=1208.573,-35.218,-40.958,179.959,5.496,148.976
C07951=1208.568,-34.968,-40.970,179.961,5.495,148.975
C07952=1208.563,-34.719,-40.983,179.964,5.496,148.974
C07953=1208.557,-34.469,-40.995,179.966,5.496,148.973
C07954=1208.552,-34.219,-41.008,179.969,5.497,148.973
C07955=1208.547,-33.969,-41.021,179.971,5.496,148.972
C07956=1208.542,-33.720,-41.033,179.974,5.497,148.971
C07957=1208.537,-33.471,-41.046,179.976,5.498,148.971
C07958=1208.532,-33.221,-41.059,179.978,5.497,148.970
C07959=1208.527,-32.971,-41.072,179.981,5.498,148.969
C07960=1208.521,-32.722,-41.085,179.983,5.498,148.969
C07961=1208.516,-32.472,-41.097,179.985,5.498,148.968
C07962=1208.511,-32.222,-41.110,179.988,5.498,148.967
C07963=1208.506,-31.972,-41.122,179.991,5.499,148.967
C07964=1208.501,-31.723,-41.135,179.993,5.499,148.966
C07965=1208.496,-31.473,-41.148,179.995,5.499,148.965
C07966=1208.491,-31.224,-41.161,179.998,5.500,148.965
C07967=1208.486,-30.974,-41.174,-180.000,5.500,148.964
C07968=1208.480,-30.725,-41.186,-179.998,5.500,148.963
C07969=1208.475,-30.475,-41.200,-179.995,5.501,148.963
C07970=1208.470,-30.225,-41.212,-179.992,5.501,148.962
C07971=1208.465,-29.976,-41.225,-179.990,5.501,148.961
C07972=1208.460,-29.726,-41.238,-179.988,5.501,148.961
C07973=1208.455,-29.476,-41.251,-179.985,5.502,148.960
C07974=1208.449,-29.227,-41.264,-179.982,5.502,148.959
C07975=1208.445,-28.977,-41.277,-179.980,5.502,148.959
C07976=1208.440,-28.728,-41.289,-179.978,5.502,148.958
C07977=1208.434,-28.478,-41.303,-179.975,5.503,148.957
C07978=1208.429,-28.228,-41.315,-179.973,5.504,148.957
C07979=1208.424,-27.979,-41.328,-179.971,5.503,148.956
C07980=1208.419,-27.729,-41.341,-179.968,5.504,148.955
C07981=1208.414,-27.479,-41.354,-179.965,5.504,148.955
C07982=1208.409,-27.230,-41.367,-179.963,5.504,148.954
C07983=1208.404,-26.981,-41.380,-179.961,5.504,148.953
C07984=1208.399,-26.731,-41.394,-179.958,5.505,148.953
C07985=1208.394,-26.481,-41.406,-179.955,5.505,148.952
C07986=1208.388,-26.232,-41.419,-179.954,5.505,148.951
C07987=1208.383,-25.982,-41.432,-179.951,5.506,148.951
C07988=1208.378,-25.732,-41.445,-179.948,5.506,148.950
C07989=1208.374,-25.482,-41.458,-179.946,5.507,148.949
C07990=1208.368,-25.233,-41.471,-179.944,5.506,148.949
C07991=1208.363,-24.983,-41.484,-179.941,5.507,148.948
C07992=1208.358,-24.734,-41.498,-179.938,5.507,148.947
C07993=1208.352,-24.484,-41.511,-179.936,5.508,148.946
C07994=1208.348,-24.234,-41.524,-179.934,5.508,148.946
C07995=1208.343,-23.985,-41.536,-179.931,5.508,148.945
C07996=1208.337,-23.735,-41.549,-179.929,5.509,148.945
C07997=1208.332,-23.485,-41.562,-179.927,5.509,148.944
C07998=1208.326,-23.217,-41.577,-179.924,5.509,148.943
C07999=1208.321,-22.947,-41.591,-179.921,5.509,148.942
C08000=1208.316,-22.678,-41.606,-179.918,5.510,148.942
C08001=1208.311,-22.408,-41.619,-179.915,5.510,148.941
C08002=1208.305,-22.158,-41.633,-179.913,5.511,148.940
C08003=1208.300,-21.909,-41.645,-179.911,5.510,148.940
C08004=1208.295,-21.659,-41.660,-179.908,5.511,148.939
C08005=1208.290,-21.410,-41.672,-179.906,5.512,148.938
C08006=1208.285,-21.159,-41.686,-179.903,5.512,148.938
C08007=1208.280,-20.910,-41.698,-179.901,5.512,148.937
C08008=1208.275,-20.661,-41.712,-179.899,5.512,148.936
C08009=1208.269,-20.411,-41.725,-179.896,5.513,148.936
C08010=1208.264,-20.162,-41.738,-179.893,5.513,148.935
C08011=1208.259,-19.912,-41.752,-179.891,5.513,148.934
C08012=1208.254,-19.663,-41.765,-179.888,5.513,148.933
C08013=1208.249,-19.412,-41.778,-179.886,5.514,148.933
C08014=1208.244,-19.163,-41.791,-179.884,5.515,148.932
C08015=1208.239,-18.913,-41.805,-179.881,5.515,148.932
C08016=1208.234,-18.664,-41.818,-179.879,5.515,148.931
C08017=1208.228,-18.414,-41.831,-179.876,5.515,148.930
C08018=1208.224,-18.165,-41.845,-179.874,5.516,148.930
C08019=1208.218,-17.915,-41.858,-179.871,5.516,148.929
C08020=1208.213,-17.665,-41.871,-179.869,5.516,148.928
C08021=1208.208,-17.416,-41.885,-179.866,5.517,148.927
C08022=1208.203,-17.166,-41.898,-179.864,5.517,148.927
C08023=1208.198,-16.917,-41.912,-179.861,5.518,148.926
C08024=1208.193,-16.667,-41.924,-179.859,5.518,148.926
C08025=1208.188,-16.417,-41.938,-179.857,5.518,148.925
C08026=1208.183,-16.168,-41.951,-179.854,5.519,148.924
C08027=1208.178,-15.918,-41.965,-179.851,5.519,148.924
C08028=1208.172,-15.669,-41.979,-179.849,5.519,148.923
C08029=1208.168,-15.419,-41.992,-179.847,5.519,148.922
C08030=1208.162,-15.170,-42.006,-179.844,5.520,148.921
C08031=1208.158,-14.920,-42.019,-179.841,5.520,148.921
C08032=1208.152,-14.670,-42.032,-179.839,5.521,148.920
C08033=1208.148,-14.421,-42.046,-179.837,5.521,148.920
C08034=1208.142,-14.171,-42.059,-179.834,5.521,148.919
C08035=1208.137,-13.922,-42.073,-179.832,5.522,148.918
C08036=1208.132,-13.672,-42.086,-179.829,5.522,148.918
C08037=1208.127,-13.423,-42.100,-179.827,5.522,148.917
C08038=1208.122,-13.173,-42.113,-179.824,5.522,148.916
C08039=1208.117,-12.924,-42.127,-179.822,5.523,148.915
C08040=1208.111,-12.673,-42.140,-179.819,5.523,148.915
C08041=1208.107,-12.425,-42.154,-179.816,5.524,148.914
C08042=1208.101,-12.174,-42.167,-179.815,5.524,148.914
C08043=1208.096,-11.925,-42.181,-179.812,5.524,148.913
C08044=1208.091,-11.676,-42.195,-179.809,5.525,148.912
C08045=1208.086,-11.425,-42.208,-179.807,5.525,148.912
C08046=1208.081,-11.177,-42.222,-179.805,5.525,148.911
C08047=1208.076,-10.926,-42.235,-179.802,5.526,148.910
C08048=1208.071,-10.677,-42.249,-179.799,5.526,148.909
C08049=1208.066,-10.427,-42.262,-179.797,5.526,148.909
C08050=1208.061,-10.178,-42.276,-179.794,5.527,148.908
C08051=1208.056,-9.929,-42.290,-179.793,5.527,148.908
C08052=1208.051,-9.679,-42.303,-179.790,5.528,148.907
C08053=1208.045,-9.430,-42.317,-179.787,5.528,148.906
C08054=1208.041,-9.180,-42.331,-179.785,5.529,148.906
C08055=1208.035,-8.930,-42.345,-179.782,5.529,148.905
C08056=1208.030,-8.681,-42.358,-179.780,5.529,148.904
C08057=1208.025,-8.431,-42.372,-179.777,5.529,148.903
C08058=1208.020,-8.182,-42.386,-179.775,5.530,148.903
C08059=1208.015,-7.932,-42.399,-179.772,5.531,148.902
C08060=1208.010,-7.682,-42.413,-179.770,5.531,148.902
C08061=1208.005,-7.433,-42.427,-179.768,5.531,148.901
C08062=1208.000,-7.183,-42.441,-179.765,5.531,148.900
C08063=1207.995,-6.934,-42.455,-179.762,5.532,148.900
C08064=1207.990,-6.684,-42.468,-179.760,5.532,148.899
C08065=1207.985,-6.434,-42.482,-179.757,5.533,148.898
C08066=1207.980,-6.185,-42.497,-179.755,5.532,148.897
C08067=1207.975,-5.935,-42.509,-179.752,5.533,148.897
C08068=1207.970,-5.686,-42.524,-179.750,5.534,148.896
C08069=1207.965,-5.436,-42.538,-179.747,5.534,148.896
C08070=1207.959,-5.187,-42.552,-179.745,5.535,148.895
C08071=1207.955,-4.937,-42.565,-179.743,5.534,148.894
C08072=1207.950,-4.687,-42.579,-179.740,5.535,148.894
C08073=1207.944,-4.438,-42.593,-179.737,5.535,148.893
C08074=1207.939,-4.188,-42.607,-179.735,5.536,148.892
C08075=1207.934,-3.939,-42.621,-179.732,5.536,148.891
C08076=1207.929,-3.689,-42.634,-179.730,5.537,148.891
C08077=1207.924,-3.440,-42.648,-179.728,5.537,148.890
C08078=1207.919,-3.190,-42.663,-179.725,5.537,148.890
C08079=1207.914,-2.941,-42.677,-179.723,5.538,148.889
C08080=1207.909,-2.691,-42.691,-179.720,5.538,148.888
C08081=1207.903,-2.441,-42.704,-179.717,5.539,148.888
C08082=1207.898,-2.191,-42.719,-179.715,5.539,148.887
C08083=1207.894,-1.943,-42.732,-179.713,5.539,148.886
C08084=1207.889,-1.693,-42.746,-179.710,5.540,148.885
C08085=1207.884,-1.443,-42.761,-179.708,5.541,148.885
C08086=1207.878,-1.194,-42.774,-179.705,5.541,148.884
C08087=1207.873,-0.944,-42.789,-179.702,5.542,148.884
C08088=1207.868,-0.695,-42.803,-179.700,5.541,148.883
C08089=1207.863,-0.444,-42.817,-179.698,5.542,148.882
C08090=1207.857,-0.195,-42.830,-179.695,5.542,148.882
C08091=1207.853,0.054,-42.844,-179.692,5.543,148.881
C08092=1207.848,0.304,-42.858,-179.690,5.543,148.880
C08093=1207.843,0.553,-42.873,-179.688,5.544,148.880
C08094=1207.838,0.802,-42.887,-179.685,5.544,148.879
C08095=1207.833,1.052,-42.901,-179.683,5.544,148.878
C08096=1207.828,1.302,-42.915,-179.680,5.545,148.878
C08097=1207.823,1.552,-42.929,-179.677,5.545,148.877
C08098=1207.817,1.801,-42.943,-179.675,5.546,148.876
C08099=1207.812,2.050,-42.958,-179.672,5.546,148.876
C08100=1207.807,2.300,-42.972,-179.670,5.547,148.875
C08101=1207.802,2.550,-42.986,-179.668,5.547,148.874
C08102=1207.797,2.819,-43.001,-179.665,5.547,148.874
C08103=1207.791,3.087,-43.016,-179.662,5.548,148.873
C08104=1207.786,3.357,-43.031,-179.660,5.548,148.872
C08105=1207.781,3.625,-43.047,-179.657,5.549,148.871
C08106=1207.776,3.875,-43.061,-179.654,5.549,148.871
C08107=1207.771,4.125,-43.076,-179.652,5.550,148.870
C08108=1207.766,4.375,-43.090,-179.649,5.550,148.870
C08109=1207.760,4.624,-43.104,-179.647,5.551,148.869
C08110=1207.755,4.873,-43.118,-179.644,5.551,148.868
C08111=1207.750,5.123,-43.132,-179.642,5.551,148.868
C08112=1207.745,5.373,-43.147,-179.639,5.552,148.867
C08113=1207.740,5.622,-43.161,-179.637,5.552,148.866
C08114=1207.735,5.872,-43.175,-179.634,5.553,148.866
C08115=1207.730,6.120,-43.190,-179.632,5.553,148.865
C08116=1207.725,6.370,-43.204,-179.629,5.554,148.864
C08117=1207.720,6.620,-43.219,-179.627,5.555,148.864
C08118=1207.715,6.870,-43.233,-179.625,5.554,148.863
C08119=1207.710,7.119,-43.247,-179.622,5.555,148.862
C08120=1207.705,7.369,-43.261,-179.619,5.555,148.862
C08121=1207.699,7.618,-43.276,-179.617,5.556,148.861
C08122=1207.694,7.867,-43.291,-179.614,5.556,148.860
C08123=1207.690,8.117,-43.305,-179.612,5.557,148.860
C08124=1207.685,8.367,-43.319,-179.609,5.558,148.859
C08125=1207.680,8.617,-43.334,-179.606,5.558,148.858
C08126=1207.675,8.866,-43.348,-179.604,5.558,148.858
C08127=1207.670,9.115,-43.363,-179.602,5.558,148.857
C08128=1207.665,9.365,-43.377,-179.599,5.559,148.856
C08129=1207.660,9.614,-43.391,-179.596,5.559,148.856
C08130=1207.655,9.864,-43.405,-179.594,5.560,148.855
C08131=1207.649,10.114,-43.420,-179.592,5.561,148.855
C08132=1207.644,10.363,-43.435,-179.589,5.561,148.854
C08133=1207.639,10.613,-43.450,-179.586,5.562,148.853
C08134=1207.634,10.862,-43.464,-179.584,5.561,148.852
C08135=1207.630,11.111,-43.479,-179.582,5.562,148.852
C08136=1207.625,11.361,-43.493,-179.579,5.562,148.851
C08137=1207.619,11.611,-43.508,-179.577,5.563,148.851
C08138=1207.614,11.861,-43.522,-179.574,5.564,148.850
C08139=1207.609,12.110,-43.537,-179.571,5.564,148.849
C08140=1207.604,12.360,-43.552,-179.569,5.565,148.849
C08141=1207.599,12.609,-43.565,-179.566,5.565,148.848
C08142=1207.594,12.858,-43.580,-179.564,5.566,148.847
C08143=1207.589,13.108,-43.595,-179.561,5.566,148.847
C08144=1207.584,13.358,-43.610,-179.559,5.566,148.846
C08145=1207.579,13.607,-43.625,-179.557,5.567,148.845
C08146=1207.574,13.856,-43.639,-179.554,5.568,148.845
C08147=1207.569,14.106,-43.653,-179.551,5.568,148.844
C08148=1207.564,14.355,-43.669,-179.549,5.569,148.843
C08149=1207.559,14.605,-43.683,-179.546,5.569,148.843
C08150=1207.554,14.854,-43.698,-179.543,5.570,148.842
C08151=1207.549,15.104,-43.712,-179.541,5.570,148.842
C08152=1207.543,15.354,-43.727,-179.539,5.571,148.841
C08153=1207.539,15.603,-43.742,-179.537,5.571,148.840
C08154=1207.534,15.853,-43.756,-179.534,5.571,148.840
C08155=1207.529,16.102,-43.771,-179.531,5.572,148.839
C08156=1207.523,16.352,-43.786,-179.529,5.572,148.838
C08157=1207.519,16.601,-43.801,-179.526,5.573,148.838
C08158=1207.514,16.851,-43.816,-179.524,5.574,148.837
C08159=1207.508,17.100,-43.831,-179.521,5.574,148.836
C08160=1207.504,17.350,-43.845,-179.518,5.575,148.836
C08161=1207.499,17.600,-43.860,-179.516,5.575,148.835
C08162=1207.494,17.849,-43.875,-179.513,5.576,148.834
C08163=1207.488,18.099,-43.890,-179.511,5.576,148.834
C08164=1207.484,18.348,-43.905,-179.509,5.576,148.833
C08165=1207.479,18.597,-43.920,-179.506,5.577,148.832
C08166=1207.473,18.847,-43.934,-179.504,5.577,148.832
C08167=1207.469,19.096,-43.949,-179.501,5.578,148.831
C08168=1207.464,19.346,-43.964,-179.498,5.578,148.830
C08169=1207.458,19.595,-43.979,-179.496,5.579,148.830
C08170=1207.453,19.845,-43.994,-179.494,5.580,148.829
C08171=1207.449,20.094,-44.009,-179.491,5.580,148.829
C08172=1207.443,20.344,-44.023,-179.488,5.581,148.828
C08173=1207.438,20.593,-44.038,-179.486,5.581,148.827
C08174=1207.433,20.842,-44.054,-179.483,5.582,148.827
C08175=1207.428,21.092,-44.068,-179.480,5.582,148.826
C08176=1207.424,21.342,-44.084,-179.479,5.582,148.825
C08177=1207.418,21.592,-44.098,-179.476,5.583,148.825
C08178=1207.414,21.841,-44.113,-179.473,5.583,148.824
C08179=1207.408,22.090,-44.129,-179.471,5.584,148.823
C08180=1207.403,22.340,-44.143,-179.468,5.584,148.823
C08181=1207.399,22.589,-44.158,-179.466,5.585,148.822
C08182=1207.393,22.839,-44.174,-179.463,5.586,148.822
C08183=1207.388,23.088,-44.188,-179.461,5.586,148.821
C08184=1207.383,23.338,-44.204,-179.458,5.587,148.820
C08185=1207.378,23.587,-44.219,-179.455,5.587,148.820
C08186=1207.372,23.837,-44.234,-179.453,5.588,148.819
C08187=1207.368,24.087,-44.249,-179.450,5.588,148.818
C08188=1207.364,24.336,-44.264,-179.448,5.589,148.818
C08189=1207.358,24.586,-44.279,-179.445,5.590,148.817
C08190=1207.353,24.835,-44.294,-179.443,5.590,148.816
C08191=1207.348,25.084,-44.309,-179.440,5.591,148.816
C08192=1207.343,25.333,-44.324,-179.437,5.591,148.815
C08193=1207.338,25.583,-44.339,-179.435,5.591,148.814
C08194=1207.333,25.832,-44.354,-179.433,5.592,148.814
C08195=1207.328,26.083,-44.370,-179.431,5.593,148.813
C08196=1207.324,26.332,-44.385,-179.428,5.593,148.813
C08197=1207.318,26.582,-44.400,-179.425,5.594,148.812
C08198=1207.313,26.831,-44.415,-179.423,5.594,148.811
C08199=1207.308,27.080,-44.431,-179.420,5.595,148.810
C08200=1207.303,27.329,-44.446,-179.418,5.596,148.810
C08201=1207.298,27.579,-44.461,-179.415,5.596,148.809
C08202=1207.294,27.829,-44.476,-179.412,5.597,148.809
C08203=1207.288,28.078,-44.492,-179.410,5.597,148.808
C08204=1207.283,28.328,-44.507,-179.407,5.598,148.807
C08205=1207.278,28.577,-44.522,-179.405,5.598,148.807
C08206=1207.273,28.845,-44.539,-179.402,5.599,148.806
C08207=1207.267,29.114,-44.555,-179.399,5.599,148.805
C08208=1207.262,29.383,-44.572,-179.397,5.600,148.805
C08209=1207.256,29.652,-44.588,-179.394,5.600,148.804
C08210=1207.252,29.902,-44.604,-179.392,5.601,148.803
C08211=1207.247,30.151,-44.619,-179.389,5.602,148.803
C08212=1207.242,30.400,-44.634,-179.387,5.602,148.802
C08213=1207.237,30.649,-44.650,-179.384,5.603,148.801
C08214=1207.231,30.899,-44.665,-179.381,5.603,148.801
C08215=1207.227,31.149,-44.681,-179.379,5.604,148.800
C08216=1207.222,31.398,-44.696,-179.376,5.605,148.800
C08217=1207.216,31.648,-44.711,-179.374,5.605,148.799
C08218=1207.211,31.897,-44.726,-179.371,5.606,148.798
C08219=1207.207,32.147,-44.742,-179.369,5.606,148.798
C08220=1207.202,32.396,-44.757,-179.366,5.607,148.797
C08221=1207.197,32.646,-44.773,-179.364,5.608,148.796
C08222=1207.191,32.895,-44.788,-179.361,5.608,148.796
C08223=1207.187,33.145,-44.804,-179.358,5.609,148.795
C08224=1207.182,33.394,-44.819,-179.356,5.609,148.794
C08225=1207.176,33.644,-44.835,-179.353,5.610,148.794
C08226=1207.172,33.893,-44.850,-179.351,5.611,148.793
C08227=1207.167,34.143,-44.866,-179.348,5.611,148.793
C08228=1207.162,34.392,-44.882,-179.346,5.612,148.792
C08229=1207.156,34.641,-44.898,-179.343,5.612,148.791
C08230=1207.152,34.890,-44.913,-179.340,5.613,148.791
C08231=1207.147,35.140,-44.929,-179.338,5.614,148.790
C08232=1207.142,35.390,-44.944,-179.336,5.614,148.789
C08233=1207.137,35.639,-44.959,-179.333,5.615,148.789
C08234=1207.132,35.888,-44.975,-179.330,5.615,148.788
C08235=1207.127,36.138,-44.991,-179.328,5.616,148.787
C08236=1207.121,36.388,-45.006,-179.326,5.617,148.787
C08237=1207.117,36.637,-45.021,-179.323,5.617,148.786
C08238=1207.112,36.887,-45.037,-179.320,5.618,148.786
C08239=1207.107,37.136,-45.053,-179.318,5.618,148.785
C08240=1207.102,37.385,-45.069,-179.315,5.619,148.784
C08241=1207.097,37.635,-45.084,-179.313,5.620,148.784
C08242=1207.092,37.884,-45.100,-179.310,5.620,148.783
C08243=1207.087,38.134,-45.116,-179.308,5.621,148.783
C08244=1207.082,38.384,-45.132,-179.305,5.621,148.782
C08245=1207.077,38.633,-45.148,-179.302,5.622,148.781
C08246=1207.072,38.882,-45.163,-179.300,5.623,148.781
C08247=1207.067,39.132,-45.179,-179.297,5.623,148.780
C08248=1207.062,39.381,-45.194,-179.295,5.624,148.779
C08249=1207.057,39.631,-45.210,-179.292,5.624,148.779
C08250=1207.052,39.880,-45.227,-179.290,5.625,148.778
C08251=1207.047,40.129,-45.242,-179.287,5.626,148.778
C08252=1207.042,40.379,-45.257,-179.285,5.626,148.777
C08253=1207.037,40.629,-45.273,-179.282,5.627,148.776
C08254=1207.032,40.877,-45.289,-179.279,5.627,148.776
C08255=1207.027,41.127,-45.305,-179.277,5.628,148.775
C08256=1207.022,41.377,-45.321,-179.275,5.629,148.774
C08257=1207.017,41.626,-45.337,-179.272,5.629,148.774
C08258=1207.013,41.876,-45.353,-179.269,5.630,148.773
C08259=1207.008,42.125,-45.368,-179.267,5.630,148.772
C08260=1207.002,42.374,-45.384,-179.265,5.631,148.772
C08261=1206.998,42.624,-45.401,-179.262,5.632,148.771
C08262=1206.992,42.873,-45.416,-179.259,5.633,148.771
C08263=1206.987,43.123,-45.432,-179.256,5.634,148.770
C08264=1206.982,43.372,-45.448,-179.253,5.634,148.769
C08265=1206.977,43.622,-45.464,-179.251,5.635,148.769
C08266=1206.972,43.872,-45.480,-179.249,5.636,148.768
C08267=1206.967,44.120,-45.496,-179.246,5.636,148.768
C08268=1206.962,44.371,-45.512,-179.243,5.637,148.767
C08269=1206.958,44.619,-45.528,-179.241,5.638,148.766
C08270=1206.953,44.868,-45.543,-179.239,5.638,148.766
C08271=1206.948,45.119,-45.559,-179.236,5.639,148.765
C08272=1206.943,45.367,-45.576,-179.233,5.639,148.764
C08273=1206.938,45.617,-45.592,-179.231,5.640,148.764
C08274=1206.933,45.866,-45.608,-179.229,5.641,148.763
C08275=1206.928,46.116,-45.624,-179.226,5.641,148.763
C08276=1206.923,46.366,-45.640,-179.223,5.642,148.762
C08277=1206.918,46.615,-45.656,-179.221,5.642,148.761
C08278=1206.913,46.865,-45.672,-179.218,5.643,148.761
C08279=1206.908,47.113,-45.688,-179.216,5.644,148.760
C08280=1206.903,47.363,-45.704,-179.213,5.644,148.759
C08281=1206.898,47.612,-45.720,-179.211,5.645,148.759
C08282=1206.893,47.862,-45.736,-179.208,5.646,148.758
C08283=1206.888,48.111,-45.753,-179.205,5.647,148.758
C08284=1206.883,48.361,-45.769,-179.203,5.648,148.757
C08285=1206.878,48.610,-45.785,-179.200,5.648,148.756
C08286=1206.873,48.860,-45.801,-179.198,5.649,148.756
C08287=1206.868,49.109,-45.817,-179.195,5.650,148.755
C08288=1206.864,49.358,-45.834,-179.193,5.650,148.755
C08289=1206.858,49.608,-45.849,-179.190,5.651,148.754
C08290=1206.854,49.857,-45.866,-179.187,5.651,148.753
C08291=1206.848,50.107,-45.882,-179.185,5.652,148.753
C08292=1206.843,50.356,-45.899,-179.182,5.653,148.752
C08293=1206.838,50.606,-45.914,-179.180,5.653,148.751
C08294=1206.834,50.855,-45.931,-179.177,5.654,148.751
C08295=1206.828,51.104,-45.947,-179.175,5.655,148.750
C08296=1206.824,51.354,-45.963,-179.172,5.655,148.750
C08297=1206.819,51.604,-45.980,-179.170,5.656,148.749
C08298=1206.814,51.852,-45.996,-179.167,5.657,148.748
C08299=1206.809,52.103,-46.012,-179.164,5.658,148.748
C08300=1206.804,52.351,-46.029,-179.162,5.659,148.747
C08301=1206.800,52.601,-46.045,-179.159,5.659,148.747
C08302=1206.794,52.851,-46.061,-179.156,5.660,148.746
C08303=1206.789,53.100,-46.078,-179.154,5.661,148.745
C08304=1206.784,53.349,-46.094,-179.152,5.661,148.745
C08305=1206.779,53.599,-46.110,-179.149,5.662,148.744
C08306=1206.775,53.848,-46.127,-179.146,5.662,148.743
C08307=1206.770,54.097,-46.143,-179.144,5.663,148.743
C08308=1206.764,54.348,-46.160,-179.142,5.664,148.742
C08309=1206.759,54.596,-46.176,-179.138,5.665,148.742
C08310=1206.754,54.865,-46.194,-179.136,5.666,148.741
C08311=1206.749,55.133,-46.211,-179.133,5.666,148.740
C08312=1206.744,55.401,-46.229,-179.131,5.667,148.740
C08313=1206.738,55.670,-46.248,-179.127,5.668,148.739
C08314=1206.733,55.920,-46.263,-179.125,5.669,148.739
C08315=1206.728,56.169,-46.280,-179.123,5.670,148.738
C08316=1206.724,56.419,-46.297,-179.120,5.670,148.737
C08317=1206.718,56.668,-46.314,-179.118,5.671,148.737
C08318=1206.713,56.918,-46.330,-179.115,5.672,148.736
C08319=1206.709,57.167,-46.346,-179.112,5.672,148.735
C08320=1206.704,57.416,-46.363,-179.110,5.673,148.735
C08321=1206.699,57.666,-46.380,-179.108,5.674,148.734
C08322=1206.693,57.915,-46.396,-179.104,5.675,148.734
C08323=1206.689,58.164,-46.413,-179.102,5.676,148.733
C08324=1206.684,58.414,-46.429,-179.099,5.676,148.732
C08325=1206.678,58.663,-46.446,-179.097,5.677,148.732
C08326=1206.674,58.913,-46.462,-179.094,5.678,148.731
C08327=1206.669,59.162,-46.479,-179.092,5.678,148.731
C08328=1206.664,59.411,-46.496,-179.090,5.679,148.730
C08329=1206.659,59.661,-46.513,-179.087,5.680,148.730
C08330=1206.655,59.910,-46.529,-179.084,5.680,148.729
C08331=1206.650,60.159,-46.545,-179.081,5.681,148.728
C08332=1206.644,60.409,-46.563,-179.079,5.682,148.728
C08333=1206.640,60.658,-46.579,-179.076,5.683,148.727
C08334=1206.635,60.907,-46.596,-179.074,5.683,148.726
C08335=1206.630,61.157,-46.613,-179.071,5.684,148.726
C08336=1206.625,61.406,-46.630,-179.069,5.685,148.725
C08337=1206.619,61.656,-46.647,-179.066,5.685,148.725
C08338=1206.615,61.905,-46.663,-179.064,5.686,148.724
C08339=1206.610,62.155,-46.680,-179.061,5.688,148.724
C08340=1206.605,62.404,-46.697,-179.058,5.688,148.723
C08341=1206.600,62.653,-46.713,-179.056,5.689,148.722
C08342=1206.595,62.903,-46.730,-179.053,5.689,148.722
C08343=1206.590,63.152,-46.747,-179.051,5.690,148.721
C08344=1206.585,63.401,-46.764,-179.048,5.691,148.720
C08345=1206.580,63.651,-46.781,-179.046,5.691,148.720
C08346=1206.575,63.900,-46.798,-179.043,5.693,148.719
C08347=1206.571,64.150,-46.814,-179.040,5.694,148.719
C08348=1206.565,64.399,-46.831,-179.038,5.694,148.718
C08349=1206.561,64.648,-46.848,-179.036,5.695,148.718
C08350=1206.555,64.898,-46.865,-179.033,5.696,148.717
C08351=1206.551,65.148,-46.882,-179.030,5.696,148.716
C08352=1206.546,65.397,-46.898,-179.028,5.697,148.716
C08353=1206.541,65.646,-46.916,-179.025,5.699,148.715
C08354=1206.537,65.895,-46.933,-179.022,5.699,148.715
C08355=1206.531,66.145,-46.950,-179.020,5.700,148.714
C08356=1206.526,66.394,-46.966,-179.018,5.701,148.713
C08357=1206.521,66.644,-46.984,-179.015,5.701,148.713
C08358=1206.517,66.893,-47.000,-179.012,5.702,148.712
C08359=1206.512,67.142,-47.018,-179.010,5.703,148.712
C08360=1206.507,67.392,-47.035,-179.007,5.704,148.711
C08361=1206.501,67.641,-47.052,-179.004,5.705,148.710
C08362=1206.497,67.890,-47.068,-179.002,5.705,148.710
C08363=1206.492,68.140,-47.086,-179.000,5.706,148.709
C08364=1206.487,68.389,-47.103,-178.997,5.707,148.709
C08365=1206.482,68.639,-47.120,-178.994,5.708,148.708
C08366=1206.477,68.888,-47.137,-178.992,5.709,148.708
C08367=1206.472,69.137,-47.154,-178.989,5.709,148.707
C08368=1206.468,69.386,-47.171,-178.986,5.710,148.706
C08369=1206.463,69.636,-47.189,-178.984,5.711,148.706
C08370=1206.458,69.885,-47.205,-178.982,5.711,148.705
C08371=1206.452,70.135,-47.222,-178.978,5.713,148.704
C08372=1206.447,70.384,-47.240,-178.976,5.714,148.704
C08373=1206.443,70.633,-47.257,-178.974,5.714,148.703
C08374=1206.438,70.883,-47.274,-178.971,5.715,148.703
C08375=1206.433,71.132,-47.291,-178.969,5.716,148.702
C08376=1206.428,71.382,-47.309,-178.966,5.716,148.702
C08377=1206.424,71.631,-47.325,-178.963,5.718,148.701
C08378=1206.418,71.880,-47.343,-178.961,5.719,148.701
C08379=1206.413,72.129,-47.360,-178.958,5.719,148.700
C08380=1206.409,72.379,-47.377,-178.956,5.720,148.699
C08381=1206.404,72.628,-47.395,-178.953,5.720,148.699
C08382=1206.398,72.878,-47.412,-178.950,5.722,148.698
C08383=1206.394,73.127,-47.429,-178.948,5.723,148.697
C08384=1206.389,73.377,-47.447,-178.945,5.723,148.697
C08385=1206.385,73.626,-47.464,-178.943,5.724,148.696
C08386=1206.379,73.875,-47.481,-178.940,5.725,148.696
C08387=1206.374,74.124,-47.498,-178.937,5.726,148.695
C08388=1206.370,74.373,-47.516,-178.935,5.727,148.695
C08389=1206.364,74.623,-47.533,-178.932,5.728,148.694
C08390=1206.359,74.873,-47.550,-178.930,5.728,148.693
C08391=1206.355,75.122,-47.568,-178.927,5.729,148.693
C08392=1206.350,75.371,-47.585,-178.924,5.730,148.692
C08393=1206.345,75.621,-47.603,-178.922,5.731,148.692
C08394=1206.340,75.870,-47.620,-178.920,5.732,148.691
C08395=1206.336,76.119,-47.638,-178.917,5.732,148.691
C08396=1206.330,76.369,-47.655,-178.915,5.733,148.690
C08397=1206.325,76.618,-47.672,-178.912,5.735,148.689
C08398=1206.320,76.867,-47.689,-178.909,5.735,148.689
C08399=1206.315,77.116,-47.707,-178.907,5.736,148.688
C08400=1206.310,77.365,-47.725,-178.904,5.737,148.688
C08401=1206.305,77.615,-47.742,-178.901,5.738,148.687
C08402=1206.301,77.864,-47.760,-178.899,5.739,148.687
C08403=1206.296,78.114,-47.777,-178.896,5.740,148.686
C08404=1206.291,78.363,-47.795,-178.894,5.740,148.685
C08405=1206.286,78.613,-47.812,-178.891,5.741,148.685
C08406=1206.282,78.862,-47.830,-178.888,5.743,148.684
C08407=1206.277,79.111,-47.848,-178.886,5.743,148.684
C08408=1206.271,79.361,-47.865,-178.883,5.744,148.683
C08409=1206.267,79.610,-47.883,-178.881,5.745,148.682
C08410=1206.261,79.860,-47.900,-178.878,5.746,148.682
C08411=1206.257,80.108,-47.918,-178.875,5.747,148.681
C08412=1206.252,80.358,-47.935,-178.873,5.748,148.681
C08413=1206.247,80.607,-47.953,-178.871,5.748,148.680
C08414=1206.242,80.876,-47.972,-178.868,5.750,148.680
C08415=1206.237,81.144,-47.992,-178.865,5.750,148.679
C08416=1206.231,81.413,-48.010,-178.862,5.751,148.678
C08417=1206.226,81.680,-48.029,-178.859,5.752,148.678
C08418=1206.221,81.930,-48.047,-178.857,5.753,148.677
C08419=1206.216,82.179,-48.065,-178.854,5.754,148.677
C08420=1206.211,82.428,-48.082,-178.851,5.755,148.676
C08421=1206.207,82.677,-48.100,-178.849,5.756,148.676
C08422=1206.201,82.927,-48.117,-178.846,5.757,148.675
C08423=1206.197,83.177,-48.136,-178.844,5.757,148.674
C08424=1206.192,83.426,-48.154,-178.841,5.759,148.674
C08425=1206.187,83.675,-48.171,-178.838,5.760,148.673
C08426=1206.182,83.925,-48.189,-178.836,5.761,148.673
C08427=1206.177,84.174,-48.207,-178.834,5.761,148.672
C08428=1206.172,84.424,-48.225,-178.830,5.762,148.671
C08429=1206.167,84.673,-48.243,-178.828,5.763,148.671
C08430=1206.163,84.922,-48.260,-178.826,5.764,148.670
C08431=1206.158,85.171,-48.277,-178.823,5.765,148.670
C08432=1206.153,85.421,-48.295,-178.820,5.766,148.669
C08433=1206.148,85.670,-48.313,-178.818,5.767,148.669
C08434=1206.143,85.919,-48.331,-178.816,5.768,148.668
C08435=1206.138,86.168,-48.349,-178.813,5.768,148.668
C08436=1206.133,86.417,-48.367,-178.810,5.770,148.667
C08437=1206.129,86.667,-48.386,-178.808,5.771,148.667
C08438=1206.124,86.916,-48.404,-178.805,5.771,148.666
C08439=1206.119,87.166,-48.421,-178.802,5.773,148.665
C08440=1206.114,87.415,-48.439,-178.800,5.774,148.665
C08441=1206.109,87.664,-48.457,-178.797,5.774,148.664
C08442=1206.104,87.914,-48.475,-178.795,5.775,148.664
C08443=1206.099,88.163,-48.493,-178.792,5.776,148.663
C08444=1206.094,88.412,-48.511,-178.789,5.777,148.662
C08445=1206.090,88.662,-48.529,-178.787,5.778,148.662
C08446=1206.085,88.911,-48.547,-178.784,5.779,148.661
C08447=1206.080,89.160,-48.565,-178.782,5.780,148.661
C08448=1206.075,89.409,-48.583,-178.779,5.781,148.660
C08449=1206.070,89.659,-48.601,-178.776,5.781,148.660
C08450=1206.065,89.908,-48.619,-178.774,5.783,148.659
C08451=1206.061,90.157,-48.637,-178.771,5.784,148.659
C08452=1206.055,90.407,-48.656,-178.769,5.785,148.658
C08453=1206.051,90.656,-48.674,-178.766,5.786,148.657
C08454=1206.046,90.905,-48.692,-178.764,5.787,148.657
C08455=1206.041,91.155,-48.710,-178.761,5.788,148.656
C08456=1206.036,91.404,-48.728,-178.758,5.788,148.656
C08457=1206.031,91.653,-48.746,-178.756,5.790,148.655
C08458=1206.027,91.903,-48.764,-178.753,5.791,148.655
C08459=1206.022,92.152,-48.782,-178.751,5.791,148.654
C08460=1206.017,92.401,-48.801,-178.748,5.793,148.654
C08461=1206.012,92.650,-48.819,-178.745,5.793,148.653
C08462=1206.007,92.899,-48.837,-178.743,5.794,148.653
C08463=1206.002,93.149,-48.856,-178.740,5.796,148.652
C08464=1205.997,93.398,-48.874,-178.738,5.797,148.652
C08465=1205.992,93.647,-48.892,-178.735,5.797,148.651
C08466=1205.987,93.897,-48.910,-178.733,5.798,148.650
C08467=1205.983,94.146,-48.928,-178.730,5.800,148.650
C08468=1205.978,94.395,-48.947,-178.727,5.800,148.649
C08469=1205.973,94.645,-48.965,-178.725,5.801,148.649
C08470=1205.968,94.894,-48.983,-178.722,5.803,148.648
C08471=1205.963,95.143,-49.001,-178.720,5.803,148.648
C08472=1205.959,95.393,-49.020,-178.717,5.804,148.647
C08473=1205.954,95.641,-49.038,-178.714,5.806,148.647
C08474=1205.949,95.891,-49.057,-178.712,5.806,148.646
C08475=1205.944,96.140,-49.075,-178.709,5.807,148.645
C08476=1205.939,96.390,-49.093,-178.706,5.809,148.645
C08477=1205.935,96.638,-49.112,-178.704,5.809,148.644
C08478=1205.929,96.888,-49.130,-178.702,5.810,148.644
C08479=1205.924,97.137,-49.148,-178.698,5.812,148.643
C08480=1205.920,97.387,-49.167,-178.696,5.813,148.643
C08481=1205.915,97.636,-49.185,-178.694,5.813,148.642
C08482=1205.910,97.885,-49.204,-178.690,5.815,148.641
C08483=1205.905,98.135,-49.222,-178.688,5.815,148.641
C08484=1205.901,98.383,-49.241,-178.686,5.816,148.640
C08485=1205.896,98.633,-49.259,-178.683,5.818,148.640
C08486=1205.890,98.882,-49.278,-178.680,5.818,148.639
C08487=1205.886,99.131,-49.297,-178.678,5.819,148.639
C08488=1205.881,99.381,-49.315,-178.675,5.821,148.638
C08489=1205.876,99.630,-49.333,-178.673,5.822,148.638
C08490=1205.872,99.879,-49.352,-178.670,5.822,148.637
C08491=1205.867,100.128,-49.370,-178.667,5.824,148.637
C08492=1205.861,100.377,-49.390,-178.665,5.825,148.636
C08493=1205.857,100.627,-49.408,-178.662,5.825,148.636
C08494=1205.852,100.876,-49.426,-178.660,5.827,148.635
C08495=1205.847,101.125,-49.445,-178.657,5.827,148.634
C08496=1205.842,101.375,-49.464,-178.655,5.828,148.634
C08497=1205.838,101.624,-49.482,-178.652,5.830,148.633
C08498=1205.832,101.873,-49.501,-178.650,5.831,148.633
C08499=1205.828,102.122,-49.520,-178.646,5.832,148.632
C08500=1205.823,102.372,-49.538,-178.644,5.833,148.632
C08501=1205.818,102.621,-49.556,-178.642,5.834,148.631
C08502=1205.814,102.870,-49.575,-178.639,5.835,148.631
C08503=1205.808,103.120,-49.594,-178.636,5.836,148.630
C08504=1205.804,103.369,-49.613,-178.634,5.837,148.630
C08505=1205.799,103.618,-49.631,-178.631,5.838,148.629
C08506=1205.794,103.867,-49.650,-178.628,5.839,148.629
C08507=1205.790,104.116,-49.669,-178.626,5.840,148.628
C08508=1205.784,104.366,-49.688,-178.623,5.841,148.628
C08509=1205.780,104.615,-49.707,-178.621,5.842,148.627
C08510=1205.774,104.865,-49.726,-178.618,5.844,148.626
C08511=1205.770,105.113,-49.744,-178.616,5.845,148.626
C08512=1205.765,105.363,-49.763,-178.613,5.845,148.625
C08513=1205.760,105.612,-49.782,-178.610,5.847,148.625
C08514=1205.756,105.861,-49.801,-178.608,5.848,148.624
C08515=1205.750,106.111,-49.820,-178.606,5.848,148.624
C08516=1205.746,106.359,-49.838,-178.602,5.850,148.623
C08517=1205.741,106.609,-49.857,-178.600,5.851,148.623
C08518=1205.735,106.877,-49.878,-178.597,5.852,148.622
C08519=1205.731,107.146,-49.898,-178.595,5.853,148.622
C08520=1205.725,107.414,-49.918,-178.592,5.855,148.621
C08521=1205.720,107.683,-49.940,-178.589,5.856,148.621
C08522=1205.715,107.932,-49.958,-178.586,5.857,148.620
C08523=1205.710,108.181,-49.977,-178.584,5.858,148.620
C08524=1205.706,108.430,-49.996,-178.581,5.859,148.619
C08525=1205.700,108.680,-50.014,-178.579,5.860,148.618
C08526=1205.696,108.929,-50.034,-178.575,5.861,148.618
C08527=1205.691,109.178,-50.053,-178.573,5.862,148.617
C08528=1205.686,109.427,-50.072,-178.571,5.863,148.617
C08529=1205.681,109.677,-50.090,-178.568,5.865,148.616
C08530=1205.677,109.926,-50.110,-178.565,5.865,148.616
C08531=1205.672,110.175,-50.129,-178.563,5.867,148.615
C08532=1205.667,110.424,-50.148,-178.560,5.868,148.615
C08533=1205.662,110.673,-50.166,-178.558,5.868,148.614
C08534=1205.658,110.923,-50.186,-178.555,5.870,148.614
C08535=1205.652,111.172,-50.205,-178.553,5.871,148.613
C08536=1205.648,111.421,-50.224,-178.549,5.872,148.613
C08537=1205.643,111.670,-50.244,-178.547,5.873,148.612
C08538=1205.638,111.920,-50.263,-178.545,5.874,148.612
C08539=1205.633,112.169,-50.281,-178.542,5.876,148.611
C08540=1205.629,112.418,-50.301,-178.539,5.876,148.611
C08541=1205.624,112.667,-50.320,-178.537,5.878,148.610
C08542=1205.619,112.916,-50.339,-178.535,5.879,148.610
C08543=1205.614,113.165,-50.359,-178.531,5.880,148.609
C08544=1205.610,113.415,-50.378,-178.529,5.881,148.609
C08545=1205.605,113.664,-50.397,-178.527,5.882,148.608
C08546=1205.599,113.914,-50.416,-178.524,5.884,148.608
C08547=1205.595,114.163,-50.436,-178.521,5.884,148.607
C08548=1205.590,114.412,-50.454,-178.519,5.886,148.607
C08549=1205.585,114.661,-50.474,-178.516,5.887,148.606
C08550=1205.580,114.910,-50.493,-178.513,5.888,148.606
C08551=1205.576,115.159,-50.512,-178.511,5.889,148.605
C08552=1205.571,115.408,-50.532,-178.509,5.890,148.605
C08553=1205.566,115.658,-50.551,-178.505,5.891,148.604
C08554=1205.561,115.907,-50.571,-178.503,5.892,148.603
C08555=1205.557,116.156,-50.590,-178.500,5.894,148.603
C08556=1205.552,116.406,-50.609,-178.498,5.895,148.602
C08557=1205.547,116.654,-50.629,-178.495,5.896,148.602
C08558=1205.542,116.904,-50.648,-178.493,5.897,148.601
C08559=1205.538,117.153,-50.667,-178.490,5.899,148.601
C08560=1205.532,117.402,-50.687,-178.487,5.899,148.600
C08561=1205.528,117.652,-50.706,-178.485,5.900,148.600
C08562=1205.522,117.901,-50.726,-178.482,5.902,148.599
C08563=1205.518,118.150,-50.745,-178.480,5.903,148.599
C08564=1205.514,118.399,-50.764,-178.477,5.904,148.598
C08565=1205.509,118.648,-50.784,-178.475,5.905,148.598
C08566=1205.504,118.897,-50.804,-178.472,5.906,148.597
C08567=1205.499,119.147,-50.824,-178.469,5.907,148.597
C08568=1205.494,119.396,-50.843,-178.467,5.909,148.596
C08569=1205.490,119.645,-50.862,-178.464,5.910,148.596
C08570=1205.485,119.894,-50.882,-178.461,5.911,148.595
C08571=1205.480,120.143,-50.901,-178.459,5.912,148.595
C08572=1205.475,120.393,-50.921,-178.456,5.914,148.594
C08573=1205.470,120.642,-50.941,-178.454,5.914,148.594
C08574=1205.465,120.891,-50.960,-178.451,5.915,148.593
C08575=1205.460,121.140,-50.980,-178.448,5.917,148.593
C08576=1205.456,121.390,-50.999,-178.446,5.918,148.592
C08577=1205.451,121.638,-51.018,-178.443,5.920,148.592
C08578=1205.447,121.887,-51.039,-178.441,5.920,148.591
C08579=1205.442,122.137,-51.058,-178.438,5.922,148.591
C08580=1205.436,122.386,-51.078,-178.435,5.923,148.590
C08581=1205.432,122.635,-51.097,-178.433,5.924,148.590
C08582=1205.427,122.884,-51.118,-178.430,5.925,148.589
C08583=1205.422,123.133,-51.137,-178.428,5.927,148.589
C08584=1205.417,123.383,-51.157,-178.425,5.928,148.588
C08585=1205.412,123.632,-51.176,-178.422,5.929,148.588
C08586=1205.408,123.881,-51.197,-178.420,5.930,148.587
C08587=1205.403,124.130,-51.216,-178.417,5.931,148.587
C08588=1205.398,124.380,-51.235,-178.415,5.932,148.586
C08589=1205.394,124.629,-51.256,-178.412,5.934,148.586
C08590=1205.390,124.878,-51.275,-178.409,5.935,148.585
C08591=1205.384,125.127,-51.294,-178.407,5.937,148.585
C08592=1205.380,125.376,-51.315,-178.404,5.937,148.584
C08593=1205.375,125.625,-51.334,-178.402,5.939,148.584
C08594=1205.370,125.875,-51.354,-178.399,5.940,148.583
C08595=1205.365,126.123,-51.374,-178.396,5.941,148.583
C08596=1205.360,126.373,-51.394,-178.394,5.942,148.582
C08597=1205.356,126.622,-51.414,-178.391,5.944,148.582
C08598=1205.351,126.872,-51.434,-178.389,5.945,148.581
C08599=1205.345,127.120,-51.453,-178.386,5.946,148.581
C08600=1205.341,127.369,-51.474,-178.384,5.947,148.580
C08601=1205.336,127.619,-51.493,-178.381,5.949,148.580
C08602=1205.332,127.868,-51.514,-178.378,5.949,148.579
C08603=1205.327,128.117,-51.534,-178.376,5.951,148.579
C08604=1205.322,128.366,-51.554,-178.373,5.952,148.578
C08605=1205.317,128.615,-51.573,-178.370,5.954,148.578
C08606=1205.313,128.864,-51.594,-178.368,5.954,148.578
C08607=1205.308,129.114,-51.613,-178.365,5.956,148.577
C08608=1205.303,129.363,-51.634,-178.363,5.957,148.577
C08609=1205.298,129.612,-51.653,-178.360,5.958,148.576
C08610=1205.294,129.861,-51.673,-178.357,5.960,148.576
C08611=1205.289,130.110,-51.693,-178.355,5.961,148.575
C08612=1205.284,130.359,-51.714,-178.352,5.962,148.575
C08613=1205.279,130.609,-51.734,-178.350,5.963,148.574
C08614=1205.275,130.858,-51.754,-178.347,5.965,148.574
C08615=1205.270,131.106,-51.774,-178.344,5.966,148.573
C08616=1205.265,131.356,-51.794,-178.342,5.968,148.573
C08617=1205.260,131.605,-51.814,-178.339,5.968,148.572
C08618=1205.256,131.854,-51.834,-178.336,5.970,148.572
C08619=1205.250,132.103,-51.855,-178.334,5.971,148.571
C08620=1205.246,132.352,-51.875,-178.331,5.972,148.571
C08621=1205.241,132.602,-51.895,-178.329,5.973,148.570
C08622=1205.236,132.870,-51.917,-178.326,5.975,148.570
C08623=1205.231,133.139,-51.938,-178.323,5.977,148.569
C08624=1205.226,133.407,-51.960,-178.320,5.978,148.569
C08625=1205.221,133.676,-51.982,-178.318,5.979,148.568
C08626=1205.216,133.925,-52.003,-178.315,5.980,148.568
C08627=1205.211,134.175,-52.022,-178.312,5.982,148.567
C08628=1205.206,134.424,-52.043,-178.310,5.983,148.567
C08629=1205.202,134.673,-52.063,-178.307,5.985,148.566
C08630=1205.197,134.922,-52.084,-178.304,5.985,148.566
C08631=1205.192,135.172,-52.104,-178.302,5.987,148.565
C08632=1205.187,135.420,-52.124,-178.299,5.988,148.565
C08633=1205.183,135.669,-52.144,-178.297,5.990,148.564
C08634=1205.177,135.918,-52.165,-178.294,5.990,148.564
C08635=1205.173,136.168,-52.185,-178.291,5.992,148.563
C08636=1205.168,136.416,-52.205,-178.289,5.994,148.563
C08637=1205.164,136.665,-52.225,-178.286,5.994,148.562
C08638=1205.159,136.915,-52.246,-178.283,5.996,148.562
C08639=1205.154,137.164,-52.267,-178.281,5.997,148.562
C08640=1205.150,137.413,-52.287,-178.278,5.999,148.561
C08641=1205.144,137.662,-52.307,-178.276,6.000,148.561
C08642=1205.140,137.911,-52.328,-178.273,6.001,148.560
C08643=1205.135,138.160,-52.348,-178.270,6.003,148.560
C08644=1205.130,138.410,-52.369,-178.268,6.004,148.559
C08645=1205.126,138.659,-52.389,-178.265,6.006,148.559
C08646=1205.121,138.908,-52.410,-178.263,6.006,148.558
C08647=1205.116,139.157,-52.431,-178.260,6.008,148.558
C08648=1205.112,139.406,-52.451,-178.257,6.010,148.557
C08649=1205.107,139.655,-52.471,-178.255,6.010,148.557
C08650=1205.102,139.905,-52.492,-178.252,6.012,148.556
C08651=1205.097,140.154,-52.512,-178.250,6.013,148.556
C08652=1205.092,140.403,-52.533,-178.247,6.015,148.555
C08653=1205.088,140.652,-52.553,-178.244,6.016,148.555
C08654=1205.083,140.901,-52.574,-178.242,6.017,148.555
C08655=1205.078,141.150,-52.595,-178.239,6.019,148.554
C08656=1205.074,141.399,-52.615,-178.237,6.020,148.554
C08657=1205.068,141.648,-52.636,-178.234,6.021,148.553
C08658=1205.064,141.897,-52.656,-178.231,6.023,148.553
C08659=1205.059,142.146,-52.677,-178.229,6.024,148.552
C08660=1205.054,142.395,-52.698,-178.226,6.026,148.552
C08661=1205.050,142.644,-52.718,-178.224,6.027,148.551
C08662=1205.045,142.893,-52.739,-178.221,6.028,148.551
C08663=1205.040,143.142,-52.759,-178.218,6.030,148.550
C08664=1205.035,143.392,-52.780,-178.216,6.031,148.550
C08665=1205.031,143.640,-52.802,-178.213,6.032,148.549
C08666=1205.026,143.889,-52.822,-178.211,6.033,148.549
C08667=1205.021,144.138,-52.843,-178.208,6.035,148.549
C08668=1205.017,144.388,-52.864,-178.205,6.036,148.548
C08669=1205.012,144.637,-52.885,-178.203,6.037,148.548
C08670=1205.007,144.886,-52.906,-178.200,6.039,148.547
C08671=1205.003,145.135,-52.926,-178.197,6.041,148.547
C08672=1204.998,145.385,-52.947,-178.195,6.042,148.546
C08673=1204.994,145.633,-52.968,-178.192,6.043,148.546
C08674=1204.988,145.882,-52.989,-178.190,6.044,148.546
C08675=1204.983,146.131,-53.010,-178.187,6.046,148.545
C08676=1204.979,146.380,-53.030,-178.184,6.048,148.545
C08677=1204.974,146.630,-53.051,-178.182,6.049,148.544
C08678=1204.970,146.879,-53.073,-178.179,6.050,148.544
C08679=1204.965,147.128,-53.094,-178.176,6.052,148.543
C08680=1204.960,147.377,-53.114,-178.174,6.053,148.543
C08681=1204.955,147.626,-53.135,-178.171,6.054,148.542
C08682=1204.950,147.875,-53.157,-178.168,6.056,148.542
C08683=1204.946,148.124,-53.177,-178.166,6.057,148.541
C08684=1204.941,148.373,-53.198,-178.163,6.059,148.541
C08685=1204.937,148.623,-53.219,-178.161,6.060,148.541
C08686=1204.932,148.871,-53.240,-178.158,6.061,148.540
C08687=1204.927,149.121,-53.261,-178.155,6.063,148.540
C08688=1204.922,149.370,-53.282,-178.153,6.064,148.539
C08689=1204.918,149.618,-53.303,-178.150,6.065,148.539
C08690=1204.912,149.867,-53.324,-178.148,6.067,148.538
C08691=1204.909,150.117,-53.345,-178.145,6.068,148.538
C08692=1204.904,150.366,-53.367,-178.143,6.070,148.537
C08693=1204.899,150.615,-53.388,-178.140,6.071,148.537
C08694=1204.894,150.864,-53.408,-178.137,6.072,148.536
C08695=1204.889,151.113,-53.430,-178.135,6.074,148.536
C08696=1204.884,151.362,-53.451,-178.132,6.076,148.536
C08697=1204.880,151.611,-53.473,-178.130,6.076,148.535
C08698=1204.875,151.860,-53.493,-178.127,6.078,148.535
C08699=1204.870,152.109,-53.514,-178.124,6.080,148.534
C08700=1204.865,152.358,-53.536,-178.122,6.081,148.534
C08701=1204.861,152.608,-53.557,-178.119,6.082,148.533
C08702=1204.857,152.856,-53.578,-178.116,6.084,148.533
C08703=1204.851,153.106,-53.599,-178.114,6.085,148.533
C08704=1204.847,153.354,-53.621,-178.111,6.087,148.532
C08705=1204.842,153.603,-53.641,-178.108,6.088,148.532
C08706=1204.838,153.852,-53.663,-178.106,6.089,148.531
C08707=1204.833,154.102,-53.684,-178.103,6.091,148.531
C08708=1204.828,154.350,-53.706,-178.101,6.093,148.530
C08709=1204.823,154.600,-53.727,-178.098,6.094,148.530
C08710=1204.819,154.849,-53.748,-178.096,6.095,148.529
C08711=1204.814,155.098,-53.769,-178.093,6.097,148.529
C08712=1204.809,155.347,-53.791,-178.090,6.099,148.529
C08713=1204.804,155.596,-53.812,-178.088,6.100,148.528
C08714=1204.800,155.845,-53.834,-178.085,6.101,148.528
C08715=1204.795,156.094,-53.855,-178.082,6.103,148.527
C08716=1204.790,156.343,-53.876,-178.080,6.104,148.527
C08717=1204.786,156.592,-53.898,-178.077,6.106,148.527
C08718=1204.781,156.841,-53.919,-178.074,6.107,148.526
C08719=1204.776,157.090,-53.941,-178.072,6.108,148.526
C08720=1204.772,157.339,-53.963,-178.070,6.110,148.525
C08721=1204.767,157.589,-53.984,-178.067,6.112,148.525
C08722=1204.762,157.837,-54.005,-178.064,6.113,148.524
C08723=1204.758,158.086,-54.027,-178.062,6.114,148.524
C08724=1204.753,158.336,-54.048,-178.059,6.116,148.524
C08725=1204.748,158.584,-54.070,-178.056,6.118,148.523
C08726=1204.743,158.854,-54.093,-178.053,6.120,148.523
C08727=1204.738,159.122,-54.117,-178.050,6.121,148.522
C08728=1204.733,159.391,-54.140,-178.048,6.122,148.522
C08729=1204.728,159.660,-54.163,-178.045,6.124,148.521
C08730=1204.723,159.909,-54.184,-178.043,6.126,148.521
C08731=1204.719,160.158,-54.206,-178.040,6.127,148.520
C08732=1204.714,160.407,-54.228,-178.037,6.129,148.520
C08733=1204.709,160.656,-54.249,-178.035,6.130,148.519
C08734=1204.705,160.906,-54.271,-178.032,6.132,148.519
C08735=1204.700,161.154,-54.293,-178.029,6.133,148.519
C08736=1204.695,161.404,-54.315,-178.027,6.134,148.518
C08737=1204.691,161.652,-54.336,-178.024,6.136,148.518
C08738=1204.685,161.901,-54.357,-178.022,6.138,148.518
C08739=1204.681,162.151,-54.379,-178.019,6.139,148.517
C08740=1204.676,162.399,-54.401,-178.017,6.140,148.517
C08741=1204.672,162.649,-54.423,-178.014,6.142,148.516
C08742=1204.667,162.897,-54.445,-178.011,6.144,148.516
C08743=1204.662,163.146,-54.467,-178.009,6.146,148.516
C08744=1204.658,163.395,-54.489,-178.006,6.146,148.515
C08745=1204.653,163.644,-54.510,-178.003,6.148,148.515
C08746=1204.648,163.894,-54.532,-178.001,6.150,148.514
C08747=1204.644,164.143,-54.553,-177.998,6.152,148.514
C08748=1204.639,164.391,-54.575,-177.996,6.153,148.513
C08749=1204.634,164.641,-54.597,-177.993,6.155,148.513
C08750=1204.630,164.889,-54.619,-177.990,6.156,148.512
C08751=1204.625,165.139,-54.641,-177.987,6.158,148.512
C08752=1204.620,165.388,-54.663,-177.985,6.159,148.512
C08753=1204.615,165.637,-54.685,-177.983,6.161,148.511
C08754=1204.611,165.886,-54.707,-177.980,6.162,148.511
C08755=1204.606,166.135,-54.729,-177.977,6.164,148.511
C08756=1204.601,166.384,-54.751,-177.975,6.165,148.510
C08757=1204.597,166.633,-54.773,-177.972,6.167,148.510
C08758=1204.592,166.882,-54.794,-177.969,6.168,148.509
C08759=1204.588,167.131,-54.816,-177.967,6.170,148.509
C08760=1204.582,167.380,-54.839,-177.964,6.172,148.509
C08761=1204.578,167.628,-54.860,-177.962,6.173,148.508
C08762=1204.574,167.877,-54.883,-177.959,6.174,148.508
C08763=1204.569,168.126,-54.905,-177.956,6.176,148.507
C08764=1204.564,168.375,-54.927,-177.953,6.178,148.507
C08765=1204.560,168.624,-54.948,-177.951,6.179,148.506
C08766=1204.555,168.873,-54.971,-177.949,6.181,148.506
C08767=1204.550,169.122,-54.993,-177.946,6.183,148.506
C08768=1204.545,169.371,-55.015,-177.943,6.184,148.505
C08769=1204.541,169.621,-55.037,-177.940,6.186,148.505
C08770=1204.536,169.869,-55.060,-177.938,6.187,148.504
C08771=1204.532,170.118,-55.082,-177.935,6.189,148.504
C08772=1204.527,170.367,-55.104,-177.933,6.190,148.504
C08773=1204.522,170.616,-55.126,-177.930,6.192,148.503
C08774=1204.518,170.865,-55.147,-177.928,6.193,148.503
C08775=1204.513,171.114,-55.171,-177.925,6.195,148.503
C08776=1204.508,171.363,-55.192,-177.922,6.197,148.502
C08777=1204.504,171.612,-55.214,-177.919,6.198,148.502
C08778=1204.498,171.861,-55.237,-177.917,6.200,148.501
C08779=1204.494,172.110,-55.259,-177.915,6.201,148.501
C08780=1204.490,172.359,-55.282,-177.912,6.203,148.500
C08781=1204.485,172.608,-55.303,-177.909,6.205,148.500
C08782=1204.480,172.857,-55.326,-177.907,6.207,148.500
C08783=1204.476,173.105,-55.348,-177.904,6.208,148.499
C08784=1204.471,173.355,-55.370,-177.901,6.209,148.499
C08785=1204.466,173.604,-55.393,-177.899,6.211,148.498
C08786=1204.462,173.852,-55.415,-177.896,6.213,148.498
C08787=1204.457,174.102,-55.437,-177.893,6.214,148.498
C08788=1204.452,174.351,-55.460,-177.891,6.216,148.497
C08789=1204.448,174.599,-55.482,-177.888,6.218,148.497
C08790=1204.444,174.849,-55.504,-177.886,6.219,148.497
C08791=1204.438,175.098,-55.527,-177.883,6.221,148.496
C08792=1204.434,175.346,-55.549,-177.881,6.223,148.496
C08793=1204.428,175.595,-55.572,-177.878,6.224,148.495
C08794=1204.424,175.844,-55.595,-177.875,6.226,148.495
C08795=1204.420,176.093,-55.617,-177.873,6.227,148.495
C08796=1204.415,176.342,-55.640,-177.870,6.229,148.494
C08797=1204.411,176.591,-55.662,-177.867,6.230,148.494
C08798=1204.406,176.841,-55.684,-177.865,6.232,148.493
C08799=1204.401,177.089,-55.707,-177.862,6.234,148.493
C08800=1204.397,177.338,-55.729,-177.859,6.236,148.493
C08801=1204.392,177.587,-55.752,-177.857,6.237,148.492
C08802=1204.387,177.836,-55.774,-177.855,6.239,148.492
C08803=1204.382,178.085,-55.797,-177.852,6.241,148.492
C08804=1204.378,178.334,-55.819,-177.849,6.242,148.491
C08805=1204.373,178.583,-55.842,-177.846,6.244,148.491
C08806=1204.369,178.831,-55.865,-177.844,6.246,148.490
C08807=1204.364,179.081,-55.888,-177.841,6.247,148.490
C08808=1204.359,179.329,-55.910,-177.839,6.248,148.490
C08809=1204.354,179.579,-55.933,-177.836,6.250,148.489
C08810=1204.350,179.827,-55.955,-177.834,6.252,148.489
C08811=1204.345,180.077,-55.978,-177.831,6.254,148.489
C08812=1204.341,180.325,-56.000,-177.828,6.256,148.488
C08813=1204.336,180.574,-56.024,-177.826,6.257,148.488
C08814=1204.332,180.823,-56.046,-177.823,6.259,148.487
C08815=1204.327,181.072,-56.069,-177.821,6.260,148.487
C08816=1204.323,181.320,-56.092,-177.818,6.262,148.487
C08817=1204.318,181.570,-56.114,-177.815,6.264,148.486
C08818=1204.314,181.819,-56.137,-177.812,6.265,148.486
C08819=1204.308,182.067,-56.160,-177.810,6.267,148.485
C08820=1204.303,182.317,-56.183,-177.807,6.269,148.485
C08821=1204.299,182.565,-56.205,-177.804,6.271,148.485
C08822=1204.295,182.815,-56.229,-177.802,6.272,148.484
C08823=1204.290,183.063,-56.250,-177.800,6.274,148.484
C08824=1204.285,183.312,-56.274,-177.797,6.275,148.484
C08825=1204.280,183.561,-56.297,-177.794,6.277,148.483
C08826=1204.276,183.810,-56.320,-177.792,6.279,148.483
C08827=1204.272,184.059,-56.343,-177.789,6.281,148.483
C08828=1204.267,184.308,-56.365,-177.786,6.283,148.482
C08829=1204.262,184.557,-56.388,-177.784,6.284,148.482
C08830=1204.257,184.826,-56.413,-177.781,6.286,148.481
C08831=1204.252,185.096,-56.438,-177.778,6.288,148.481
C08832=1204.247,185.366,-56.463,-177.775,6.290,148.481
C08833=1204.242,185.635,-56.488,-177.772,6.291,148.480
C08834=1204.238,185.884,-56.511,-177.770,6.293,148.480
C08835=1204.233,186.133,-56.534,-177.767,6.295,148.479
C08836=1204.228,186.382,-56.557,-177.765,6.297,148.479
C08837=1204.224,186.631,-56.580,-177.762,6.299,148.479
C08838=1204.219,186.879,-56.603,-177.759,6.300,148.478
C08839=1204.214,187.128,-56.626,-177.757,6.301,148.478
C08840=1204.210,187.377,-56.649,-177.754,6.303,148.478
C08841=1204.206,187.626,-56.673,-177.752,6.305,148.477
C08842=1204.201,187.876,-56.695,-177.749,6.307,148.477
C08843=1204.196,188.125,-56.719,-177.746,6.309,148.477
C08844=1204.191,188.373,-56.741,-177.744,6.310,148.476
C08845=1204.187,188.622,-56.764,-177.741,6.312,148.476
C08846=1204.182,188.871,-56.788,-177.739,6.314,148.476
C08847=1204.177,189.120,-56.811,-177.736,6.316,148.475
C08848=1204.173,189.369,-56.834,-177.733,6.318,148.475
C08849=1204.169,189.618,-56.857,-177.731,6.320,148.475
C08850=1204.164,189.867,-56.881,-177.728,6.321,148.474
C08851=1204.159,190.116,-56.904,-177.726,6.322,148.474
C08852=1204.155,190.365,-56.927,-177.723,6.324,148.473
C08853=1204.149,190.613,-56.950,-177.720,6.326,148.473
C08854=1204.146,190.861,-56.974,-177.718,6.328,148.473
C08855=1204.141,191.110,-56.997,-177.715,6.330,148.472
C08856=1204.136,191.359,-57.020,-177.713,6.331,148.472
C08857=1204.131,191.608,-57.044,-177.710,6.333,148.472
C08858=1204.127,191.857,-57.067,-177.707,6.335,148.471
C08859=1204.122,192.106,-57.091,-177.705,6.337,148.471
C08860=1204.117,192.355,-57.114,-177.702,6.339,148.471
C08861=1204.113,192.604,-57.137,-177.699,6.341,148.470
C08862=1204.109,192.853,-57.160,-177.697,6.342,148.470
C08863=1204.104,193.101,-57.184,-177.694,6.344,148.470
C08864=1204.100,193.350,-57.207,-177.691,6.346,148.469
C08865=1204.095,193.600,-57.231,-177.689,6.348,148.469
C08866=1204.090,193.849,-57.254,-177.687,6.349,148.469
C08867=1204.086,194.098,-57.278,-177.684,6.351,148.468
C08868=1204.081,194.345,-57.301,-177.681,6.352,148.468
C08869=1204.076,194.594,-57.325,-177.679,6.354,148.468
C08870=1204.071,194.843,-57.348,-177.676,6.356,148.467
C08871=1204.066,195.092,-57.371,-177.673,6.358,148.467
C08872=1204.062,195.341,-57.395,-177.671,6.360,148.466
C08873=1204.057,195.590,-57.419,-177.668,6.362,148.466
C08874=1204.053,195.839,-57.442,-177.665,6.363,148.466
C08875=1204.048,196.088,-57.465,-177.663,6.365,148.465
C08876=1204.044,196.336,-57.490,-177.660,6.367,148.465
C08877=1204.039,196.585,-57.513,-177.657,6.369,148.465
C08878=1204.034,196.834,-57.536,-177.655,6.371,148.464
C08879=1204.030,197.083,-57.560,-177.652,6.372,148.464
C08880=1204.025,197.332,-57.584,-177.649,6.374,148.464
C08881=1204.021,197.582,-57.607,-177.647,6.376,148.463
C08882=1204.017,197.830,-57.631,-177.644,6.378,148.463
C08883=1204.012,198.079,-57.655,-177.641,6.380,148.463
C08884=1204.007,198.327,-57.679,-177.639,6.382,148.462
C08885=1204.003,198.576,-57.702,-177.636,6.383,148.462
C08886=1203.998,198.825,-57.726,-177.633,6.385,148.462
C08887=1203.994,199.074,-57.750,-177.631,6.387,148.462
C08888=1203.989,199.323,-57.773,-177.629,6.389,148.461
C08889=1203.985,199.571,-57.797,-177.626,6.391,148.461
C08890=1203.980,199.820,-57.820,-177.623,6.393,148.460
C08891=1203.975,200.069,-57.845,-177.621,6.395,148.460
C08892=1203.971,200.318,-57.868,-177.618,6.396,148.460
C08893=1203.966,200.566,-57.892,-177.615,6.398,148.459
C08894=1203.961,200.816,-57.916,-177.613,6.400,148.459
C08895=1203.957,201.064,-57.940,-177.610,6.402,148.459
C08896=1203.952,201.314,-57.964,-177.607,6.404,148.458
C08897=1203.948,201.562,-57.988,-177.605,6.406,148.458
C08898=1203.943,201.811,-58.011,-177.602,6.407,148.458
C08899=1203.939,202.060,-58.035,-177.599,6.409,148.457
C08900=1203.934,202.309,-58.059,-177.597,6.411,148.457
C08901=1203.929,202.557,-58.083,-177.594,6.413,148.457
C08902=1203.925,202.806,-58.107,-177.592,6.415,148.457
C08903=1203.920,203.055,-58.131,-177.589,6.417,148.456
C08904=1203.916,203.304,-58.155,-177.587,6.419,148.456
C08905=1203.912,203.553,-58.179,-177.584,6.420,148.456
C08906=1203.906,203.802,-58.203,-177.581,6.422,148.455
C08907=1203.902,204.050,-58.227,-177.579,6.424,148.455
C08908=1203.897,204.299,-58.251,-177.576,6.426,148.455
C08909=1203.893,204.547,-58.275,-177.573,6.428,148.454
C08910=1203.889,204.796,-58.299,-177.571,6.430,148.454
C08911=1203.884,205.046,-58.323,-177.568,6.431,148.454
C08912=1203.879,205.294,-58.347,-177.566,6.433,148.453
C08913=1203.875,205.543,-58.371,-177.563,6.435,148.453
C08914=1203.871,205.791,-58.395,-177.561,6.437,148.453
C08915=1203.865,206.041,-58.419,-177.558,6.439,148.452
C08916=1203.861,206.290,-58.444,-177.555,6.441,148.452
C08917=1203.857,206.538,-58.468,-177.553,6.443,148.452
C08918=1203.852,206.787,-58.492,-177.550,6.445,148.451
C08919=1203.847,207.036,-58.516,-177.547,6.446,148.451
C08920=1203.843,207.284,-58.540,-177.545,6.448,148.451
C08921=1203.838,207.534,-58.565,-177.542,6.450,148.450
C08922=1203.834,207.782,-58.589,-177.540,6.452,148.450
C08923=1203.829,208.030,-58.613,-177.537,6.454,148.450
C08924=1203.824,208.280,-58.637,-177.535,6.456,148.450
C08925=1203.820,208.528,-58.661,-177.532,6.458,148.449
C08926=1203.816,208.777,-58.686,-177.529,6.459,148.449
C08927=1203.811,209.026,-58.710,-177.527,6.461,148.449
C08928=1203.806,209.274,-58.734,-177.524,6.463,148.448
C08929=1203.802,209.523,-58.758,-177.521,6.465,148.448
C08930=1203.797,209.772,-58.783,-177.518,6.468,148.448
C08931=1203.793,210.021,-58.807,-177.516,6.470,148.447
C08932=1203.788,210.269,-58.832,-177.513,6.472,148.447
C08933=1203.783,210.518,-58.855,-177.511,6.473,148.447
C08934=1203.778,210.789,-58.883,-177.508,6.475,148.446
C08935=1203.773,211.060,-58.909,-177.506,6.477,148.446
C08936=1203.768,211.330,-58.936,-177.502,6.480,148.446
C08937=1203.764,211.600,-58.962,-177.500,6.482,148.445
C08938=1203.759,211.849,-58.987,-177.497,6.483,148.445
C08939=1203.755,212.097,-59.011,-177.494,6.485,148.445
C08940=1203.750,212.346,-59.036,-177.492,6.487,148.444
C08941=1203.746,212.595,-59.060,-177.489,6.489,148.444
C08942=1203.741,212.844,-59.085,-177.486,6.491,148.444
C08943=1203.736,213.092,-59.109,-177.484,6.493,148.444
C08944=1203.732,213.342,-59.134,-177.481,6.496,148.443
C08945=1203.727,213.590,-59.158,-177.478,6.497,148.443
C08946=1203.722,213.839,-59.183,-177.476,6.499,148.443
C08947=1203.719,214.088,-59.207,-177.473,6.501,148.442
C08948=1203.713,214.337,-59.232,-177.471,6.503,148.442
C08949=1203.709,214.585,-59.256,-177.468,6.505,148.442
C08950=1203.704,214.835,-59.281,-177.466,6.507,148.442
C08951=1203.700,215.082,-59.306,-177.463,6.509,148.441
C08952=1203.695,215.331,-59.331,-177.460,6.510,148.441
C08953=1203.691,215.580,-59.355,-177.458,6.512,148.441
C08954=1203.686,215.829,-59.380,-177.455,6.514,148.440
C08955=1203.681,216.078,-59.404,-177.453,6.516,148.440
C08956=1203.677,216.327,-59.429,-177.450,6.519,148.440
C08957=1203.673,216.575,-59.454,-177.447,6.521,148.439
C08958=1203.669,216.824,-59.479,-177.444,6.523,148.439
C08959=1203.664,217.073,-59.503,-177.442,6.524,148.439
C08960=1203.659,217.321,-59.528,-177.439,6.526,148.438
C08961=1203.655,217.570,-59.553,-177.437,6.528,148.438
C08962=1203.650,217.819,-59.578,-177.434,6.530,148.438
C08963=1203.646,218.068,-59.602,-177.432,6.532,148.438
C08964=1203.641,218.316,-59.628,-177.429,6.534,148.437
C08965=1203.636,218.565,-59.652,-177.426,6.537,148.437
C08966=1203.632,218.814,-59.677,-177.424,6.539,148.437
C08967=1203.627,219.062,-59.701,-177.421,6.541,148.437
C08968=1203.623,219.311,-59.727,-177.418,6.542,148.436
C08969=1203.619,219.560,-59.751,-177.416,6.544,148.436
C08970=1203.614,219.808,-59.777,-177.413,6.546,148.436
C08971=1203.609,220.057,-59.802,-177.411,6.548,148.436
C08972=1203.605,220.307,-59.827,-177.408,6.550,148.435
C08973=1203.601,220.554,-59.851,-177.406,6.552,148.435
C08974=1203.596,220.803,-59.876,-177.403,6.555,148.435
C08975=1203.591,221.053,-59.901,-177.400,6.556,148.434
C08976=1203.587,221.300,-59.926,-177.398,6.559,148.434
C08977=1203.582,221.550,-59.951,-177.395,6.560,148.434
C08978=1203.578,221.798,-59.976,-177.392,6.562,148.433
C08979=1203.573,222.047,-60.001,-177.390,6.564,148.433
C08980=1203.569,222.295,-60.026,-177.387,6.566,148.433
C08981=1203.564,222.545,-60.051,-177.385,6.568,148.433
C08982=1203.560,222.793,-60.077,-177.382,6.570,148.432
C08983=1203.555,223.042,-60.102,-177.379,6.573,148.432
C08984=1203.550,223.290,-60.127,-177.377,6.574,148.432
C08985=1203.546,223.539,-60.151,-177.374,6.577,148.432
C08986=1203.542,223.787,-60.177,-177.372,6.578,148.431
C08987=1203.537,224.037,-60.202,-177.369,6.580,148.431
C08988=1203.532,224.285,-60.227,-177.366,6.582,148.431
C08989=1203.528,224.534,-60.252,-177.364,6.584,148.431
C08990=1203.524,224.783,-60.277,-177.361,6.587,148.430
C08991=1203.519,225.031,-60.303,-177.358,6.589,148.430
C08992=1203.515,225.280,-60.328,-177.356,6.591,148.430
C08993=1203.510,225.528,-60.353,-177.354,6.593,148.429
C08994=1203.506,225.777,-60.379,-177.351,6.595,148.429
C08995=1203.501,226.026,-60.404,-177.348,6.596,148.429
C08996=1203.496,226.275,-60.429,-177.346,6.598,148.429
C08997=1203.491,226.524,-60.454,-177.343,6.601,148.428
C08998=1203.488,226.772,-60.479,-177.340,6.603,148.428
C08999=1203.484,227.021,-60.505,-177.338,6.605,148.428
C09000=1203.479,227.269,-60.530,-177.335,6.607,148.427
C09001=1203.474,227.518,-60.555,-177.333,6.609,148.427
C09002=1203.469,227.766,-60.581,-177.330,6.611,148.427
C09003=1203.465,228.015,-60.607,-177.328,6.613,148.427
C09004=1203.461,228.265,-60.632,-177.325,6.616,148.427
C09005=1203.456,228.513,-60.657,-177.322,6.617,148.426
C09006=1203.452,228.762,-60.683,-177.320,6.619,148.426
C09007=1203.447,229.010,-60.708,-177.317,6.621,148.426
C09008=1203.443,229.258,-60.734,-177.315,6.623,148.426
C09009=1203.438,229.508,-60.759,-177.312,6.625,148.425
C09010=1203.433,229.756,-60.784,-177.309,6.628,148.425
C09011=1203.429,230.005,-60.810,-177.307,6.630,148.425
C09012=1203.425,230.254,-60.836,-177.304,6.632,148.425
C09013=1203.420,230.502,-60.861,-177.302,6.634,148.424
C09014=1203.416,230.751,-60.887,-177.299,6.636,148.424
C09015=1203.411,230.999,-60.912,-177.297,6.638,148.424
C09016=1203.406,231.248,-60.937,-177.294,6.640,148.423
C09017=1203.402,231.497,-60.963,-177.291,6.642,148.423
C09018=1203.397,231.745,-60.988,-177.289,6.644,148.423
C09019=1203.393,231.994,-61.014,-177.286,6.646,148.423
C09020=1203.389,232.243,-61.040,-177.284,6.648,148.422
C09021=1203.385,232.491,-61.066,-177.281,6.650,148.422
C09022=1203.380,232.739,-61.091,-177.278,6.653,148.422
C09023=1203.376,232.988,-61.117,-177.276,6.655,148.422
C09024=1203.371,233.237,-61.143,-177.273,6.657,148.422
C09025=1203.366,233.486,-61.169,-177.271,6.659,148.421
C09026=1203.362,233.734,-61.194,-177.268,6.661,148.421
C09027=1203.357,233.983,-61.220,-177.265,6.663,148.421
C09028=1203.353,234.231,-61.245,-177.263,6.665,148.421
C09029=1203.348,234.480,-61.271,-177.260,6.667,148.420
C09030=1203.344,234.729,-61.297,-177.258,6.669,148.420
C09031=1203.340,234.978,-61.323,-177.255,6.671,148.420
C09032=1203.334,235.226,-61.349,-177.253,6.673,148.419
C09033=1203.330,235.475,-61.374,-177.250,6.676,148.419
C09034=1203.326,235.724,-61.400,-177.247,6.678,148.419
C09035=1203.322,235.972,-61.426,-177.245,6.680,148.419
C09036=1203.317,236.221,-61.451,-177.243,6.682,148.419
C09037=1203.312,236.470,-61.478,-177.240,6.684,148.418
C09038=1203.307,236.741,-61.506,-177.237,6.686,148.418
C09039=1203.302,237.012,-61.534,-177.234,6.688,148.418
C09040=1203.298,237.283,-61.563,-177.231,6.691,148.417
C09041=1203.293,237.555,-61.591,-177.229,6.693,148.417
C09042=1203.288,237.803,-61.616,-177.226,6.696,148.417
C09043=1203.283,238.053,-61.643,-177.223,6.698,148.417
C09044=1203.279,238.301,-61.669,-177.221,6.700,148.417
C09045=1203.275,238.550,-61.695,-177.218,6.702,148.416
C09046=1203.271,238.798,-61.721,-177.215,6.705,148.416
C09047=1203.265,239.047,-61.747,-177.213,6.707,148.416
C09048=1203.261,239.295,-61.773,-177.210,6.708,148.416
C09049=1203.257,239.544,-61.799,-177.208,6.711,148.416
C09050=1203.252,239.793,-61.825,-177.205,6.712,148.415
C09051=1203.248,240.042,-61.851,-177.202,6.715,148.415
C09052=1203.244,240.290,-61.877,-177.200,6.717,148.415
C09053=1203.239,240.538,-61.903,-177.197,6.719,148.415
C09054=1203.234,240.787,-61.929,-177.195,6.721,148.414
C09055=1203.230,241.035,-61.956,-177.192,6.724,148.414
C09056=1203.226,241.284,-61.981,-177.189,6.726,148.414
C09057=1203.221,241.533,-62.008,-177.187,6.728,148.414
C09058=1203.217,241.781,-62.034,-177.185,6.730,148.413
C09059=1203.212,242.030,-62.060,-177.182,6.733,148.413
C09060=1203.207,242.279,-62.086,-177.179,6.735,148.413
C09061=1203.204,242.527,-62.112,-177.177,6.737,148.413
C09062=1203.199,242.776,-62.139,-177.175,6.739,148.413
C09063=1203.195,243.024,-62.165,-177.172,6.741,148.412
C09064=1203.190,243.273,-62.191,-177.169,6.744,148.412
C09065=1203.186,243.521,-62.218,-177.167,6.745,148.412
C09066=1203.182,243.770,-62.244,-177.164,6.747,148.412
C09067=1203.176,244.018,-62.270,-177.162,6.749,148.412
C09068=1203.172,244.267,-62.296,-177.159,6.752,148.411
C09069=1203.167,244.515,-62.323,-177.156,6.754,148.411
C09070=1203.163,244.764,-62.349,-177.154,6.756,148.411
C09071=1203.159,245.013,-62.376,-177.151,6.758,148.411
C09072=1203.154,245.261,-62.402,-177.149,6.761,148.410
C09073=1203.150,245.510,-62.429,-177.146,6.763,148.410
C09074=1203.145,245.759,-62.455,-177.144,6.765,148.410
C09075=1203.142,246.007,-62.481,-177.141,6.768,148.410
C09076=1203.137,246.256,-62.507,-177.138,6.770,148.410
C09077=1203.133,246.504,-62.534,-177.136,6.772,148.409
C09078=1203.128,246.753,-62.561,-177.134,6.774,148.409
C09079=1203.123,247.002,-62.587,-177.130,6.777,148.409
C09080=1203.119,247.250,-62.614,-177.128,6.778,148.409
C09081=1203.114,247.499,-62.640,-177.126,6.781,148.409
C09082=1203.110,247.747,-62.667,-177.123,6.782,148.408
C09083=1203.106,247.996,-62.694,-177.120,6.785,148.408
C09084=1203.101,248.244,-62.719,-177.118,6.787,148.408
C09085=1203.096,248.492,-62.746,-177.116,6.789,148.408
C09086=1203.092,248.741,-62.773,-177.112,6.792,148.408
C09087=1203.087,248.990,-62.799,-177.110,6.794,148.407
C09088=1203.083,249.238,-62.826,-177.108,6.796,148.407
C09089=1203.079,249.486,-62.852,-177.105,6.798,148.407
C09090=1203.074,249.735,-62.879,-177.102,6.801,148.407
C09091=1203.070,249.984,-62.905,-177.100,6.803,148.406
C09092=1203.065,250.232,-62.932,-177.097,6.805,148.406
C09093=1203.061,250.481,-62.960,-177.094,6.808,148.406
C09094=1203.057,250.730,-62.986,-177.092,6.810,148.406
C09095=1203.052,250.978,-63.013,-177.090,6.812,148.406
C09096=1203.048,251.227,-63.040,-177.087,6.814,148.406
C09097=1203.044,251.475,-63.066,-177.084,6.817,148.405
C09098=1203.039,251.724,-63.093,-177.082,6.819,148.405
C09099=1203.034,251.972,-63.120,-177.079,6.821,148.405
C09100=1203.030,252.220,-63.147,-177.077,6.824,148.405
C09101=1203.026,252.469,-63.174,-177.074,6.825,148.405
C09102=1203.021,252.718,-63.200,-177.072,6.828,148.405
C09103=1203.017,252.966,-63.226,-177.069,6.830,148.404
C09104=1203.012,253.215,-63.254,-177.067,6.832,148.404
C09105=1203.008,253.463,-63.281,-177.064,6.834,148.404
C09106=1203.003,253.712,-63.308,-177.061,6.837,148.404
C09107=1202.999,253.960,-63.334,-177.059,6.839,148.403
C09108=1202.994,254.208,-63.361,-177.056,6.841,148.403
C09109=1202.990,254.457,-63.388,-177.053,6.844,148.403
C09110=1202.986,254.706,-63.415,-177.051,6.846,148.403
C09111=1202.982,254.954,-63.442,-177.049,6.848,148.403
C09112=1202.977,255.203,-63.469,-177.046,6.851,148.403
C09113=1202.972,255.451,-63.496,-177.043,6.853,148.402
C09114=1202.968,255.700,-63.523,-177.041,6.855,148.402
C09115=1202.964,255.948,-63.550,-177.038,6.857,148.402
C09116=1202.959,256.196,-63.577,-177.036,6.860,148.402
C09117=1202.954,256.445,-63.604,-177.033,6.862,148.402
C09118=1202.950,256.694,-63.631,-177.030,6.865,148.402
C09119=1202.946,256.943,-63.658,-177.028,6.867,148.401
C09120=1202.941,257.191,-63.685,-177.026,6.869,148.401
C09121=1202.937,257.439,-63.712,-177.023,6.872,148.401
C09122=1202.933,257.687,-63.740,-177.020,6.874,148.401
C09123=1202.928,257.936,-63.767,-177.018,6.876,148.401
C09124=1202.923,258.184,-63.794,-177.015,6.879,148.400
C09125=1202.919,258.433,-63.821,-177.013,6.881,148.400
C09126=1202.915,258.682,-63.848,-177.010,6.883,148.400
C09127=1202.910,258.930,-63.875,-177.007,6.886,148.400
C09128=1202.906,259.178,-63.903,-177.005,6.887,148.400
C09129=1202.902,259.426,-63.930,-177.003,6.890,148.400
C09130=1202.898,259.676,-63.957,-177.000,6.892,148.399
C09131=1202.893,259.924,-63.984,-176.997,6.895,148.399
C09132=1202.888,260.173,-64.011,-176.995,6.897,148.399
C09133=1202.884,260.421,-64.039,-176.992,6.899,148.399
C09134=1202.879,260.669,-64.066,-176.990,6.902,148.399
